C03638=1033.348,389.943,360.918,173.337,46.298,159.226
C03639=1033.357,390.188,360.876,173.346,46.301,159.228
C03640=1033.366,390.434,360.834,173.354,46.305,159.230
C03641=1033.376,390.680,360.790,173.364,46.308,159.232
C03642=1033.385,390.926,360.747,173.373,46.312,159.234
C03643=1033.394,391.173,360.704,173.381,46.316,159.236
C03644=1033.403,391.418,360.661,173.390,46.319,159.238
C03645=1033.413,391.665,360.617,173.399,46.323,159.240
C03646=1033.421,391.911,360.574,173.408,46.326,159.242
C03647=1033.431,392.156,360.531,173.417,46.330,159.244
C03648=1033.440,392.402,360.488,173.426,46.334,159.246
C03649=1033.450,392.649,360.445,173.435,46.337,159.248
C03650=1033.458,392.881,360.404,173.443,46.341,159.250
C03651=1033.467,393.113,360.362,173.452,46.345,159.252
C03652=1033.476,393.346,360.321,173.460,46.348,159.254
C03653=1033.485,393.578,360.281,173.469,46.352,159.256
C03654=1033.494,393.811,360.240,173.477,46.355,159.258
C03655=1033.502,394.044,360.198,173.486,46.359,159.260
C03656=1033.511,394.277,360.158,173.495,46.363,159.262
C03657=1033.521,394.509,360.116,173.505,46.366,159.264
C03658=1033.530,394.756,360.073,173.513,46.370,159.266
C03659=1033.539,395.001,360.029,173.522,46.374,159.268
C03660=1033.548,395.247,359.985,173.532,46.377,159.270
C03661=1033.558,395.493,359.941,173.541,46.381,159.272
C03662=1033.568,395.739,359.897,173.551,46.385,159.274
C03663=1033.577,395.984,359.854,173.560,46.389,159.276
C03664=1033.587,396.230,359.810,173.569,46.393,159.278
C03665=1033.596,396.476,359.766,173.578,46.397,159.280
C03666=1033.606,396.723,359.722,173.587,46.401,159.282
C03667=1033.614,396.968,359.678,173.597,46.405,159.285
C03668=1033.625,397.214,359.635,173.606,46.409,159.287
C03669=1033.634,397.460,359.590,173.616,46.413,159.289
C03670=1033.644,397.705,359.546,173.626,46.416,159.291
C03671=1033.654,397.951,359.502,173.635,46.421,159.293
C03672=1033.663,398.197,359.458,173.645,46.424,159.296
C03673=1033.673,398.443,359.413,173.654,46.429,159.298
C03674=1033.682,398.689,359.369,173.664,46.433,159.300
C03675=1033.692,398.935,359.326,173.673,46.437,159.302
C03676=1033.702,399.180,359.281,173.683,46.441,159.304
C03677=1033.712,399.427,359.237,173.693,46.445,159.307
C03678=1033.721,399.672,359.192,173.702,46.449,159.309
C03679=1033.731,399.918,359.148,173.712,46.453,159.311
C03680=1033.740,400.164,359.103,173.722,46.457,159.313
C03681=1033.751,400.410,359.059,173.731,46.462,159.316
C03682=1033.760,400.655,359.015,173.742,46.466,159.318
C03683=1033.770,400.901,358.970,173.752,46.470,159.320
C03684=1033.780,401.146,358.925,173.761,46.475,159.323
C03685=1033.790,401.393,358.880,173.771,46.479,159.325
C03686=1033.799,401.638,358.836,173.781,46.483,159.327
C03687=1033.809,401.884,358.791,173.791,46.487,159.330
C03688=1033.819,402.129,358.746,173.802,46.491,159.332
C03689=1033.829,402.375,358.701,173.811,46.496,159.334
C03690=1033.839,402.621,358.656,173.821,46.500,159.337
C03691=1033.849,402.867,358.611,173.831,46.505,159.339
C03692=1033.858,403.112,358.566,173.841,46.508,159.341
C03693=1033.867,403.358,358.521,173.852,46.513,159.344
C03694=1033.878,403.604,358.475,173.861,46.518,159.346
C03695=1033.888,403.849,358.430,173.871,46.522,159.348
C03696=1033.897,404.095,358.385,173.882,46.527,159.351
C03697=1033.908,404.341,358.340,173.892,46.531,159.353
C03698=1033.918,404.586,358.295,173.902,46.535,159.356
C03699=1033.928,404.832,358.249,173.913,46.540,159.358
C03700=1033.937,405.078,358.204,173.923,46.544,159.361
C03701=1033.947,405.323,358.158,173.933,46.549,159.363
C03702=1033.957,405.569,358.113,173.944,46.553,159.365
C03703=1033.967,405.814,358.068,173.954,46.558,159.368
C03704=1033.978,406.060,358.023,173.965,46.563,159.371
C03705=1033.988,406.306,357.976,173.975,46.567,159.373
C03706=1033.997,406.551,357.931,173.985,46.572,159.375
C03707=1034.008,406.797,357.885,173.996,46.576,159.378
C03708=1034.018,407.042,357.840,174.006,46.581,159.380
C03709=1034.029,407.287,357.794,174.017,46.585,159.383
C03710=1034.039,407.531,357.749,174.027,46.590,159.386
C03711=1034.049,407.773,357.704,174.038,46.595,159.388
C03712=1034.059,408.017,357.658,174.048,46.599,159.390
C03713=1034.069,408.259,357.613,174.059,46.604,159.393
C03714=1034.079,408.503,357.568,174.069,46.609,159.396
C03715=1034.089,408.745,357.523,174.080,46.614,159.398
C03716=1034.100,408.988,357.477,174.091,46.618,159.401
C03717=1034.110,409.231,357.431,174.102,46.623,159.403
C03718=1034.121,409.476,357.385,174.112,46.628,159.406
C03719=1034.130,409.722,357.339,174.123,46.633,159.409
C03720=1034.141,409.967,357.293,174.134,46.638,159.411
C03721=1034.151,410.213,357.247,174.145,46.642,159.414
C03722=1034.162,410.458,357.201,174.156,46.647,159.416
C03723=1034.172,410.704,357.154,174.166,46.652,159.419
C03724=1034.183,410.949,357.108,174.178,46.656,159.422
C03725=1034.193,411.195,357.062,174.189,46.662,159.424
C03726=1034.204,411.440,357.015,174.200,46.667,159.427
C03727=1034.214,411.686,356.969,174.211,46.671,159.430
C03728=1034.224,411.931,356.922,174.222,46.676,159.432
C03729=1034.235,412.176,356.876,174.234,46.681,159.435
C03730=1034.245,412.422,356.829,174.245,46.686,159.438
C03731=1034.257,412.668,356.782,174.255,46.691,159.441
C03732=1034.267,412.913,356.735,174.267,46.697,159.444
C03733=1034.277,413.159,356.689,174.278,46.701,159.446
C03734=1034.288,413.404,356.642,174.290,46.707,159.449
C03735=1034.298,413.649,356.594,174.301,46.712,159.452
C03736=1034.309,413.894,356.548,174.313,46.717,159.455
C03737=1034.320,414.140,356.500,174.325,46.722,159.458
C03738=1034.331,414.385,356.454,174.336,46.727,159.460
C03739=1034.341,414.630,356.406,174.347,46.732,159.463
C03740=1034.352,414.875,356.360,174.358,46.738,159.466
C03741=1034.362,415.121,356.312,174.370,46.743,159.469
C03742=1034.373,415.366,356.266,174.382,46.748,159.472
C03743=1034.384,415.612,356.218,174.393,46.753,159.475
C03744=1034.395,415.857,356.171,174.405,46.758,159.477
C03745=1034.406,416.102,356.123,174.417,46.764,159.480
C03746=1034.417,416.348,356.076,174.429,46.769,159.483
C03747=1034.427,416.593,356.029,174.441,46.774,159.486
C03748=1034.438,416.838,355.981,174.453,46.780,159.489
C03749=1034.449,417.083,355.934,174.465,46.785,159.492
C03750=1034.460,417.329,355.887,174.477,46.790,159.495
C03751=1034.471,417.574,355.839,174.488,46.796,159.498
C03752=1034.482,417.819,355.791,174.500,46.801,159.501
C03753=1034.493,418.064,355.744,174.513,46.807,159.504
C03754=1034.504,418.309,355.696,174.525,46.812,159.507
C03755=1034.514,418.554,355.648,174.537,46.818,159.510
C03756=1034.525,418.800,355.599,174.549,46.823,159.513
C03757=1034.537,419.045,355.552,174.561,46.829,159.516
C03758=1034.547,419.290,355.504,174.574,46.834,159.519
C03759=1034.558,419.535,355.456,174.586,46.840,159.522
C03760=1034.570,419.781,355.408,174.598,46.846,159.525
C03761=1034.581,420.026,355.360,174.610,46.851,159.528
C03762=1034.591,420.271,355.312,174.623,46.856,159.531
C03763=1034.603,420.515,355.263,174.635,46.862,159.535
C03764=1034.614,420.760,355.215,174.647,46.868,159.538
C03765=1034.625,421.006,355.167,174.660,46.874,159.541
C03766=1034.637,421.251,355.118,174.672,46.880,159.544
C03767=1034.648,421.497,355.070,174.685,46.885,159.547
C03768=1034.660,421.741,355.022,174.697,46.891,159.550
C03769=1034.670,421.986,354.974,174.711,46.897,159.554
C03770=1034.682,422.236,354.924,174.723,46.902,159.557
C03771=1034.693,422.485,354.874,174.736,46.909,159.560
C03772=1034.706,422.735,354.825,174.750,46.915,159.564
C03773=1034.717,422.985,354.775,174.762,46.920,159.567
C03774=1034.728,423.230,354.726,174.776,46.926,159.570
C03775=1034.739,423.475,354.678,174.788,46.932,159.573
C03776=1034.751,423.720,354.629,174.801,46.938,159.576
C03777=1034.762,423.965,354.580,174.814,46.944,159.580
C03778=1034.774,424.210,354.531,174.827,46.950,159.583
C03779=1034.786,424.455,354.482,174.840,46.956,159.587
C03780=1034.797,424.700,354.433,174.854,46.962,159.590
C03781=1034.809,424.944,354.384,174.866,46.968,159.593
C03782=1034.820,425.189,354.335,174.880,46.974,159.597
C03783=1034.832,425.434,354.285,174.893,46.980,159.600
C03784=1034.843,425.679,354.236,174.906,46.986,159.603
C03785=1034.854,425.924,354.187,174.919,46.992,159.607
C03786=1034.866,426.169,354.137,174.933,46.998,159.610
C03787=1034.878,426.414,354.088,174.947,47.004,159.614
C03788=1034.889,426.659,354.039,174.960,47.011,159.617
C03789=1034.901,426.903,353.988,174.974,47.016,159.621
C03790=1034.913,427.148,353.939,174.988,47.023,159.624
C03791=1034.925,427.394,353.890,175.000,47.029,159.627
C03792=1034.937,427.638,353.840,175.014,47.035,159.631
C03793=1034.948,427.883,353.790,175.028,47.042,159.635
C03794=1034.960,428.128,353.740,175.042,47.047,159.638
C03795=1034.972,428.372,353.691,175.055,47.054,159.642
C03796=1034.984,428.617,353.640,175.069,47.060,159.645
C03797=1034.995,428.862,353.590,175.083,47.067,159.649
C03798=1035.007,429.106,353.540,175.097,47.073,159.652
C03799=1035.019,429.351,353.490,175.111,47.079,159.656
C03800=1035.031,429.596,353.440,175.126,47.086,159.660
C03801=1035.043,429.841,353.390,175.140,47.092,159.663
C03802=1035.055,430.085,353.339,175.154,47.099,159.667
C03803=1035.066,430.330,353.289,175.168,47.105,159.671
C03804=1035.079,430.574,353.238,175.182,47.112,159.674
C03805=1035.091,430.819,353.188,175.196,47.118,159.678
C03806=1035.104,431.064,353.138,175.211,47.125,159.682
C03807=1035.115,431.308,353.087,175.225,47.132,159.686
C03808=1035.128,431.553,353.037,175.239,47.138,159.689
C03809=1035.140,431.796,352.986,175.254,47.145,159.693
C03810=1035.151,432.042,352.935,175.268,47.152,159.697
C03811=1035.164,432.286,352.885,175.284,47.158,159.701
C03812=1035.176,432.531,352.835,175.298,47.164,159.704
C03813=1035.188,432.775,352.783,175.312,47.171,159.708
C03814=1035.201,433.020,352.732,175.327,47.178,159.712
C03815=1035.214,433.265,352.682,175.342,47.185,159.716
C03816=1035.226,433.509,352.631,175.357,47.192,159.720
C03817=1035.238,433.754,352.580,175.372,47.198,159.724
C03818=1035.251,433.998,352.529,175.386,47.205,159.727
C03819=1035.264,434.243,352.478,175.402,47.212,159.732
C03820=1035.276,434.487,352.426,175.417,47.219,159.735
C03821=1035.289,434.731,352.375,175.432,47.226,159.739
C03822=1035.301,434.975,352.323,175.447,47.232,159.743
C03823=1035.314,435.220,352.272,175.463,47.239,159.747
C03824=1035.326,435.465,352.221,175.477,47.247,159.751
C03825=1035.339,435.708,352.169,175.493,47.253,159.755
C03826=1035.351,435.954,352.117,175.508,47.260,159.759
C03827=1035.364,436.197,352.066,175.523,47.267,159.763
C03828=1035.376,436.442,352.015,175.539,47.274,159.767
C03829=1035.390,436.686,351.963,175.555,47.281,159.772
C03830=1035.402,436.935,351.909,175.571,47.289,159.776
C03831=1035.415,437.183,351.857,175.587,47.296,159.780
C03832=1035.428,437.432,351.805,175.603,47.303,159.784
C03833=1035.441,437.680,351.751,175.619,47.310,159.788
C03834=1035.454,437.924,351.700,175.634,47.318,159.793
C03835=1035.466,438.169,351.647,175.650,47.325,159.797
C03836=1035.479,438.413,351.595,175.666,47.332,159.801
C03837=1035.492,438.657,351.543,175.682,47.339,159.805
C03838=1035.505,438.901,351.490,175.698,47.347,159.810
C03839=1035.519,439.145,351.438,175.714,47.354,159.814
C03840=1035.532,439.390,351.386,175.731,47.361,159.818
C03841=1035.544,439.633,351.333,175.747,47.369,159.822
C03842=1035.558,439.877,351.281,175.764,47.376,159.827
C03843=1035.570,440.122,351.228,175.780,47.384,159.831
C03844=1035.583,440.366,351.175,175.796,47.391,159.835
C03845=1035.597,440.609,351.123,175.812,47.398,159.840
C03846=1035.610,440.854,351.070,175.829,47.406,159.844
C03847=1035.623,441.098,351.017,175.846,47.413,159.849
C03848=1035.636,441.342,350.964,175.862,47.421,159.853
C03849=1035.650,441.585,350.911,175.879,47.428,159.857
C03850=1035.663,441.829,350.858,175.896,47.436,159.862
C03851=1035.676,442.073,350.805,175.913,47.444,159.867
C03852=1035.689,442.317,350.751,175.930,47.451,159.871
C03853=1035.703,442.561,350.699,175.947,47.458,159.875
C03854=1035.717,442.806,350.645,175.963,47.466,159.880
C03855=1035.730,443.050,350.592,175.981,47.474,159.885
C03856=1035.743,443.293,350.538,175.999,47.482,159.889
C03857=1035.757,443.537,350.486,176.015,47.490,159.894
C03858=1035.771,443.780,350.432,176.033,47.497,159.899
C03859=1035.785,444.023,350.378,176.050,47.505,159.903
C03860=1035.799,444.267,350.326,176.067,47.513,159.908
C03861=1035.813,444.510,350.274,176.085,47.520,159.912
C03862=1035.828,444.753,350.221,176.102,47.528,159.917
C03863=1035.844,444.996,350.169,176.121,47.535,159.922
C03864=1035.861,445.240,350.118,176.138,47.542,159.926
C03865=1035.877,445.484,350.067,176.156,47.550,159.931
C03866=1035.894,445.727,350.017,176.174,47.557,159.935
C03867=1035.913,445.971,349.967,176.191,47.564,159.940
C03868=1035.931,446.215,349.918,176.210,47.571,159.944
C03869=1035.949,446.460,349.869,176.228,47.577,159.949
C03870=1035.969,446.704,349.820,176.247,47.584,159.954
C03871=1035.989,446.948,349.772,176.265,47.591,159.958
C03872=1036.009,447.193,349.724,176.283,47.598,159.963
C03873=1036.031,447.437,349.677,176.301,47.604,159.967
C03874=1036.052,447.681,349.630,176.320,47.611,159.971
C03875=1036.075,447.926,349.583,176.339,47.617,159.976
C03876=1036.097,448.170,349.538,176.357,47.623,159.980
C03877=1036.120,448.415,349.492,176.376,47.629,159.985
C03878=1036.144,448.660,349.447,176.395,47.636,159.989
C03879=1036.168,448.905,349.402,176.414,47.642,159.994
C03880=1036.192,449.150,349.359,176.434,47.648,159.998
C03881=1036.218,449.395,349.314,176.452,47.653,160.002
C03882=1036.244,449.640,349.271,176.471,47.659,160.007
C03883=1036.271,449.885,349.228,176.492,47.665,160.011
C03884=1036.297,450.130,349.185,176.510,47.670,160.016
C03885=1036.325,450.376,349.144,176.531,47.676,160.020
C03886=1036.352,450.621,349.102,176.549,47.682,160.024
C03887=1036.382,450.866,349.061,176.569,47.687,160.029
C03888=1036.410,451.112,349.020,176.589,47.692,160.033
C03889=1036.440,451.357,348.980,176.609,47.698,160.037
C03890=1036.473,451.633,348.935,176.631,47.703,160.042
C03891=1036.509,451.908,348.891,176.654,47.709,160.047
C03892=1036.544,452.183,348.848,176.677,47.715,160.052
C03893=1036.579,452.458,348.805,176.699,47.720,160.057
C03894=1036.290,452.515,348.480,176.702,47.790,160.079
C03895=1036.256,452.253,348.521,176.681,47.785,160.074
C03896=1036.222,451.991,348.562,176.659,47.780,160.070
C03897=1036.188,451.729,348.604,176.638,47.775,160.065
C03898=1036.157,451.467,348.646,176.616,47.769,160.060
C03899=1036.127,451.222,348.686,176.596,47.764,160.056
C03900=1036.097,450.976,348.726,176.576,47.759,160.052
C03901=1036.068,450.730,348.768,176.557,47.754,160.047
C03902=1036.040,450.484,348.809,176.537,47.748,160.043
C03903=1036.012,450.240,348.850,176.517,47.743,160.039
C03904=1035.985,449.995,348.893,176.498,47.737,160.034
C03905=1035.958,449.750,348.936,176.478,47.732,160.030
C03906=1035.932,449.504,348.979,176.459,47.726,160.026
C03907=1035.907,449.259,349.022,176.440,47.720,160.021
C03908=1035.881,449.014,349.066,176.421,47.715,160.017
C03909=1035.857,448.769,349.111,176.402,47.709,160.012
C03910=1035.833,448.524,349.156,176.383,47.703,160.008
C03911=1035.810,448.279,349.201,176.363,47.697,160.003
C03912=1035.786,448.034,349.246,176.344,47.690,159.999
C03913=1035.764,447.790,349.292,176.326,47.684,159.994
C03914=1035.742,447.546,349.339,176.307,47.678,159.990
C03915=1035.721,447.302,349.386,176.289,47.671,159.986
C03916=1035.700,447.057,349.433,176.270,47.665,159.981
C03917=1035.680,446.812,349.481,176.251,47.659,159.977
C03918=1035.660,446.569,349.530,176.233,47.652,159.972
C03919=1035.641,446.324,349.578,176.215,47.645,159.968
C03920=1035.622,446.080,349.628,176.197,47.638,159.963
C03921=1035.604,445.836,349.678,176.179,47.631,159.958
C03922=1035.587,445.593,349.728,176.160,47.624,159.954
C03923=1035.569,445.349,349.778,176.143,47.618,159.949
C03924=1035.553,445.104,349.829,176.125,47.610,159.945
C03925=1035.537,444.861,349.881,176.107,47.603,159.940
C03926=1035.521,444.618,349.933,176.089,47.596,159.936
C03927=1035.506,444.374,349.985,176.072,47.588,159.931
C03928=1035.491,444.131,350.037,176.054,47.581,159.926
C03929=1035.477,443.888,350.090,176.037,47.573,159.922
C03930=1035.464,443.646,350.143,176.020,47.565,159.917
C03931=1035.450,443.402,350.197,176.002,47.557,159.912
C03932=1035.436,443.158,350.251,175.985,47.550,159.908
C03933=1035.423,442.914,350.304,175.967,47.542,159.903
C03934=1035.410,442.670,350.357,175.951,47.535,159.899
C03935=1035.396,442.426,350.410,175.933,47.528,159.894
C03936=1035.383,442.181,350.464,175.917,47.520,159.890
C03937=1035.369,441.938,350.517,175.899,47.512,159.885
C03938=1035.356,441.694,350.569,175.883,47.504,159.881
C03939=1035.343,441.450,350.623,175.866,47.497,159.876
C03940=1035.330,441.206,350.676,175.849,47.490,159.872
C03941=1035.316,440.962,350.728,175.832,47.483,159.867
C03942=1035.303,440.718,350.782,175.816,47.475,159.863
C03943=1035.290,440.474,350.834,175.800,47.468,159.859
C03944=1035.277,440.230,350.887,175.782,47.460,159.854
C03945=1035.263,439.986,350.940,175.766,47.453,159.850
C03946=1035.251,439.742,350.992,175.750,47.446,159.845
C03947=1035.238,439.498,351.045,175.733,47.438,159.841
C03948=1035.224,439.254,351.097,175.718,47.431,159.837
C03949=1035.211,439.009,351.150,175.700,47.424,159.833
C03950=1035.199,438.765,351.202,175.684,47.417,159.828
C03951=1035.185,438.520,351.254,175.668,47.409,159.824
C03952=1035.173,438.277,351.307,175.652,47.403,159.820
C03953=1035.159,438.033,351.359,175.636,47.395,159.815
C03954=1035.146,437.788,351.411,175.620,47.388,159.811
C03955=1035.134,437.539,351.464,175.604,47.381,159.807
C03956=1035.120,437.290,351.517,175.588,47.374,159.803
C03957=1035.107,437.040,351.570,175.572,47.366,159.799
C03958=1035.095,436.790,351.623,175.556,47.360,159.795
C03959=1035.081,436.546,351.675,175.541,47.353,159.790
C03960=1035.069,436.302,351.727,175.525,47.346,159.786
C03961=1035.056,436.057,351.778,175.510,47.339,159.782
C03962=1035.044,435.813,351.830,175.494,47.332,159.778
C03963=1035.031,435.569,351.881,175.478,47.325,159.774
C03964=1035.018,435.324,351.933,175.463,47.318,159.770
C03965=1035.006,435.080,351.984,175.448,47.311,159.766
C03966=1034.994,434.836,352.036,175.432,47.304,159.762
C03967=1034.980,434.591,352.087,175.418,47.297,159.758
C03968=1034.968,434.347,352.139,175.402,47.290,159.754
C03969=1034.956,434.103,352.190,175.388,47.284,159.750
C03970=1034.943,433.857,352.241,175.372,47.277,159.746
C03971=1034.931,433.612,352.292,175.358,47.270,159.743
C03972=1034.918,433.368,352.342,175.342,47.264,159.739
C03973=1034.906,433.124,352.393,175.328,47.257,159.735
C03974=1034.894,432.880,352.445,175.312,47.251,159.731
C03975=1034.881,432.635,352.496,175.298,47.244,159.727
C03976=1034.869,432.391,352.546,175.284,47.237,159.723
C03977=1034.857,432.146,352.597,175.268,47.231,159.719
C03978=1034.844,431.902,352.648,175.254,47.224,159.716
C03979=1034.832,431.657,352.698,175.240,47.218,159.712
C03980=1034.820,431.413,352.749,175.225,47.211,159.708
C03981=1034.808,431.168,352.799,175.211,47.205,159.705
C03982=1034.795,430.923,352.850,175.196,47.198,159.701
C03983=1034.783,430.679,352.900,175.181,47.192,159.697
C03984=1034.771,430.434,352.951,175.167,47.185,159.693
C03985=1034.760,430.189,353.001,175.153,47.179,159.690
C03986=1034.747,429.945,353.051,175.139,47.172,159.686
C03987=1034.736,429.699,353.102,175.125,47.166,159.682
C03988=1034.724,429.456,353.152,175.111,47.160,159.679
C03989=1034.711,429.211,353.202,175.096,47.153,159.675
C03990=1034.699,428.966,353.251,175.082,47.147,159.671
C03991=1034.688,428.721,353.302,175.068,47.141,159.668
C03992=1034.676,428.476,353.352,175.054,47.135,159.664
C03993=1034.664,428.232,353.402,175.041,47.128,159.661
C03994=1034.653,427.987,353.452,175.027,47.122,159.657
C03995=1034.640,427.742,353.502,175.013,47.115,159.654
C03996=1034.629,427.498,353.551,174.999,47.110,159.650
C03997=1034.617,427.253,353.601,174.985,47.103,159.647
C03998=1034.605,427.008,353.651,174.973,47.097,159.643
C03999=1034.593,426.763,353.701,174.958,47.091,159.640
C04000=1034.582,426.518,353.750,174.945,47.085,159.636
C04001=1034.570,426.273,353.800,174.932,47.079,159.633
C04002=1034.559,426.029,353.849,174.918,47.073,159.629
C04003=1034.547,425.784,353.898,174.904,47.067,159.626
C04004=1034.535,425.538,353.948,174.891,47.061,159.622
C04005=1034.524,425.294,353.997,174.878,47.055,159.619
C04006=1034.512,425.049,354.046,174.865,47.049,159.616
C04007=1034.501,424.804,354.095,174.851,47.043,159.612
C04008=1034.489,424.559,354.144,174.838,47.037,159.609
C04009=1034.478,424.314,354.193,174.825,47.031,159.606
C04010=1034.466,424.069,354.242,174.812,47.025,159.602
C04011=1034.455,423.825,354.291,174.799,47.020,159.599
C04012=1034.443,423.580,354.340,174.786,47.013,159.596
C04013=1034.432,423.335,354.389,174.774,47.008,159.593
C04014=1034.421,423.090,354.437,174.760,47.002,159.589
C04015=1034.409,422.838,354.488,174.747,46.996,159.586
C04016=1034.397,422.586,354.538,174.733,46.990,159.583
C04017=1034.385,422.333,354.588,174.720,46.985,159.579
C04018=1034.373,422.082,354.637,174.707,46.978,159.576
C04019=1034.362,421.837,354.686,174.695,46.973,159.573
C04020=1034.351,421.592,354.735,174.681,46.967,159.569
C04021=1034.340,421.346,354.783,174.669,46.961,159.566
C04022=1034.328,421.102,354.832,174.656,46.956,159.563
C04023=1034.317,420.857,354.880,174.644,46.950,159.560
C04024=1034.306,420.611,354.928,174.632,46.944,159.557
C04025=1034.294,420.366,354.976,174.619,46.939,159.554
C04026=1034.283,420.120,355.024,174.607,46.933,159.551
C04027=1034.273,419.876,355.072,174.594,46.928,159.548
C04028=1034.262,419.630,355.121,174.581,46.923,159.545
C04029=1034.250,419.385,355.168,174.569,46.917,159.541
C04030=1034.239,419.140,355.217,174.557,46.911,159.538
C04031=1034.228,418.895,355.265,174.545,46.906,159.535
C04032=1034.217,418.650,355.313,174.532,46.901,159.532
C04033=1034.207,418.405,355.361,174.520,46.895,159.529
C04034=1034.195,418.160,355.409,174.509,46.889,159.526
C04035=1034.184,417.914,355.456,174.497,46.884,159.523
C04036=1034.174,417.670,355.504,174.484,46.879,159.520
C04037=1034.162,417.424,355.552,174.472,46.874,159.517
C04038=1034.152,417.179,355.600,174.460,46.868,159.514
C04039=1034.140,416.934,355.647,174.448,46.863,159.511
C04040=1034.130,416.689,355.694,174.436,46.858,159.508
C04041=1034.119,416.443,355.741,174.425,46.852,159.506
C04042=1034.108,416.197,355.789,174.413,46.847,159.503
C04043=1034.097,415.953,355.836,174.401,46.842,159.500
C04044=1034.087,415.707,355.884,174.389,46.837,159.497
C04045=1034.075,415.462,355.931,174.377,46.832,159.494
C04046=1034.065,415.216,355.978,174.366,46.826,159.491
C04047=1034.054,414.970,356.025,174.354,46.822,159.488
C04048=1034.043,414.725,356.072,174.342,46.816,159.485
C04049=1034.033,414.481,356.120,174.331,46.811,159.483
C04050=1034.022,414.235,356.166,174.319,46.806,159.480
C04051=1034.011,413.989,356.213,174.308,46.801,159.477
C04052=1034.000,413.744,356.260,174.296,46.796,159.474
C04053=1033.990,413.499,356.307,174.285,46.791,159.471
C04054=1033.979,413.254,356.354,174.273,46.786,159.468
C04055=1033.969,413.009,356.401,174.262,46.781,159.466
C04056=1033.957,412.763,356.448,174.251,46.775,159.463
C04057=1033.947,412.517,356.495,174.239,46.771,159.460
C04058=1033.937,412.272,356.541,174.228,46.766,159.458
C04059=1033.926,412.027,356.588,174.216,46.761,159.455
C04060=1033.916,411.781,356.634,174.206,46.756,159.452
C04061=1033.906,411.536,356.682,174.195,46.751,159.449
C04062=1033.895,411.290,356.727,174.183,46.746,159.447
C04063=1033.885,411.045,356.775,174.173,46.741,159.444
C04064=1033.874,410.799,356.821,174.161,46.737,159.441
C04065=1033.863,410.554,356.866,174.150,46.732,159.439
C04066=1033.854,410.308,356.913,174.139,46.727,159.436
C04067=1033.843,410.063,356.960,174.128,46.722,159.433
C04068=1033.832,409.817,357.005,174.117,46.717,159.431
C04069=1033.821,409.572,357.051,174.106,46.712,159.428
C04070=1033.811,409.326,357.097,174.095,46.708,159.425
C04071=1033.801,409.083,357.143,174.084,46.703,159.423
C04072=1033.791,408.838,357.189,174.074,46.699,159.420
C04073=1033.781,408.595,357.234,174.063,46.694,159.418
C04074=1033.770,408.350,357.280,174.053,46.689,159.415
C04075=1033.760,408.107,357.326,174.041,46.685,159.413
C04076=1033.750,407.863,357.371,174.031,46.680,159.410
C04077=1033.739,407.619,357.416,174.020,46.675,159.407
C04078=1033.730,407.375,357.462,174.010,46.671,159.405
C04079=1033.719,407.129,357.507,173.999,46.667,159.403
C04080=1033.709,406.884,357.553,173.989,46.662,159.400
C04081=1033.699,406.639,357.599,173.978,46.657,159.397
C04082=1033.688,406.392,357.644,173.968,46.653,159.395
C04083=1033.679,406.147,357.690,173.957,46.649,159.393
C04084=1033.669,405.901,357.735,173.946,46.644,159.390
C04085=1033.659,405.656,357.781,173.936,46.639,159.387
C04086=1033.648,405.410,357.826,173.925,46.635,159.385
C04087=1033.638,405.165,357.872,173.915,46.630,159.383
C04088=1033.628,404.919,357.917,173.905,46.626,159.380
C04089=1033.619,404.674,357.963,173.894,46.621,159.378
C04090=1033.608,404.427,358.008,173.884,46.617,159.375
C04091=1033.599,404.182,358.053,173.875,46.613,159.373
C04092=1033.588,403.936,358.099,173.864,46.608,159.371
C04093=1033.578,403.691,358.144,173.854,46.604,159.368
C04094=1033.569,403.445,358.189,173.844,46.599,159.366
C04095=1033.560,403.199,358.234,173.833,46.595,159.363
C04096=1033.549,402.953,358.279,173.823,46.591,159.361
C04097=1033.540,402.708,358.324,173.813,46.587,159.359
C04098=1033.530,402.462,358.369,173.803,46.582,159.356
C04099=1033.520,402.216,358.414,173.794,46.578,159.354
C04100=1033.510,401.970,358.459,173.783,46.574,159.351
C04101=1033.500,401.725,358.504,173.773,46.570,159.349
C04102=1033.490,401.479,358.549,173.763,46.566,159.347
C04103=1033.481,401.234,358.593,173.753,46.561,159.345
C04104=1033.471,400.988,358.638,173.744,46.557,159.342
C04105=1033.461,400.742,358.683,173.734,46.553,159.340
C04106=1033.451,400.496,358.727,173.723,46.549,159.338
C04107=1033.441,400.251,358.772,173.713,46.545,159.335
C04108=1033.431,400.005,358.816,173.704,46.541,159.333
C04109=1033.422,399.759,358.861,173.694,46.537,159.331
C04110=1033.412,399.514,358.905,173.684,46.532,159.329
C04111=1033.403,399.268,358.950,173.675,46.528,159.326
C04112=1033.393,399.022,358.994,173.665,46.524,159.324
C04113=1033.383,398.776,359.038,173.655,46.520,159.322
C04114=1033.373,398.530,359.082,173.646,46.516,159.320
C04115=1033.364,398.285,359.127,173.636,46.513,159.318
C04116=1033.354,398.038,359.171,173.626,46.509,159.315
C04117=1033.344,397.793,359.214,173.617,46.505,159.313
C04118=1033.335,397.547,359.259,173.607,46.501,159.311
C04119=1033.325,397.301,359.303,173.598,46.496,159.309
C04120=1033.315,397.056,359.347,173.588,46.493,159.307
C04121=1033.306,396.810,359.391,173.578,46.489,159.305
C04122=1033.297,396.564,359.435,173.569,46.485,159.302
C04123=1033.286,396.318,359.478,173.559,46.481,159.300
C04124=1033.277,396.072,359.522,173.551,46.477,159.298
C04125=1033.268,395.826,359.566,173.541,46.473,159.296
C04126=1033.259,395.580,359.610,173.532,46.470,159.294
C04127=1033.249,395.334,359.654,173.522,46.466,159.292
C04128=1033.239,395.088,359.698,173.513,46.462,159.290
C04129=1033.230,394.843,359.742,173.504,46.458,159.287
C04130=1033.220,394.597,359.785,173.495,46.455,159.285
C04131=1033.212,394.363,359.826,173.486,46.451,159.283
C04132=1033.203,394.129,359.868,173.477,46.447,159.281
C04133=1033.194,393.895,359.910,173.468,46.444,159.279
C04134=1033.184,393.661,359.950,173.460,46.441,159.278
C04135=1033.176,393.428,359.992,173.451,46.437,159.276
C04136=1033.167,393.195,360.033,173.443,46.433,159.274
C04137=1033.158,392.960,360.074,173.434,46.430,159.272
C04138=1033.149,392.727,360.115,173.425,46.426,159.270
C04139=1033.140,392.481,360.159,173.416,46.423,159.268
C04140=1033.130,392.235,360.202,173.407,46.419,159.266
C04141=1033.121,391.989,360.245,173.398,46.416,159.264
C04142=1033.112,391.743,360.288,173.389,46.412,159.262
C04143=1033.103,391.497,360.332,173.380,46.409,159.260
C04144=1033.093,391.251,360.374,173.371,46.405,159.258
C04145=1033.084,391.005,360.417,173.362,46.402,159.256
C04146=1033.074,390.759,360.461,173.353,46.398,159.254
C04147=1033.066,390.513,360.504,173.344,46.394,159.252
C04148=1033.057,390.267,360.546,173.335,46.391,159.250
C04149=1033.047,390.020,360.590,173.327,46.387,159.248
C04150=1033.038,389.775,360.632,173.317,46.384,159.246
C04151=1033.028,389.528,360.675,173.309,46.380,159.244
C04152=1033.020,389.282,360.718,173.300,46.377,159.242
C04153=1033.011,389.036,360.760,173.292,46.374,159.240
C04154=1033.001,388.790,360.803,173.283,46.370,159.239
C04155=1032.992,388.544,360.846,173.274,46.367,159.236
C04156=1032.983,388.298,360.889,173.265,46.363,159.235
C04157=1032.975,388.052,360.932,173.256,46.360,159.233
C04158=1032.965,387.806,360.975,173.248,46.357,159.231
C04159=1032.956,387.560,361.017,173.239,46.353,159.229
C04160=1032.947,387.313,361.059,173.231,46.350,159.227
C04161=1032.938,387.067,361.102,173.222,46.347,159.225
C04162=1032.928,386.821,361.145,173.214,46.343,159.223
C04163=1032.919,386.575,361.186,173.206,46.340,159.222
C04164=1032.910,386.329,361.229,173.196,46.337,159.220
C04165=1032.901,386.082,361.270,173.187,46.334,159.218
C04166=1032.892,385.837,361.313,173.179,46.331,159.216
C04167=1032.883,385.590,361.355,173.171,46.327,159.214
C04168=1032.873,385.344,361.397,173.162,46.324,159.212
C04169=1032.865,385.097,361.440,173.154,46.321,159.211
C04170=1032.856,384.851,361.481,173.146,46.318,159.209
C04171=1032.847,384.605,361.524,173.137,46.315,159.207
C04172=1032.838,384.359,361.566,173.129,46.312,159.205
C04173=1032.829,384.112,361.607,173.120,46.309,159.203
C04174=1032.820,383.867,361.650,173.112,46.305,159.202
C04175=1032.811,383.620,361.691,173.104,46.302,159.200
C04176=1032.802,383.374,361.733,173.095,46.299,159.198
C04177=1032.793,383.128,361.775,173.087,46.296,159.196
C04178=1032.784,382.881,361.817,173.080,46.293,159.195
C04179=1032.775,382.635,361.858,173.071,46.290,159.193
C04180=1032.766,382.389,361.901,173.063,46.287,159.191
C04181=1032.757,382.143,361.942,173.055,46.284,159.189
C04182=1032.748,381.896,361.984,173.047,46.281,159.188
C04183=1032.740,381.650,362.026,173.038,46.278,159.186
C04184=1032.731,381.404,362.068,173.030,46.275,159.184
C04185=1032.722,381.158,362.109,173.022,46.272,159.183
C04186=1032.714,380.911,362.150,173.014,46.269,159.181
C04187=1032.705,380.664,362.192,173.006,46.266,159.179
C04188=1032.696,380.418,362.234,172.998,46.263,159.178
C04189=1032.688,380.172,362.275,172.990,46.260,159.176
C04190=1032.679,379.926,362.317,172.982,46.257,159.174
C04191=1032.671,379.709,362.353,172.974,46.255,159.173
C04192=1032.664,379.493,362.390,172.968,46.252,159.171
C04193=1032.656,379.277,362.426,172.961,46.249,159.170
C04194=1032.648,379.061,362.463,172.954,46.247,159.168
C04195=1032.640,378.845,362.498,172.947,46.244,159.167
C04196=1032.634,378.629,362.535,172.940,46.242,159.165
C04197=1032.626,378.413,362.572,172.933,46.239,159.164
C04198=1032.618,378.196,362.607,172.926,46.237,159.163
C04199=1032.610,377.950,362.649,172.918,46.234,159.161
C04200=1032.601,377.704,362.690,172.911,46.231,159.159
C04201=1032.592,377.457,362.731,172.903,46.228,159.158
C04202=1032.584,377.211,362.772,172.895,46.226,159.156
C04203=1032.575,376.964,362.812,172.888,46.223,159.154
C04204=1032.566,376.718,362.854,172.879,46.220,159.153
C04205=1032.558,376.472,362.895,172.871,46.218,159.151
C04206=1032.548,376.225,362.935,172.863,46.215,159.150
C04207=1032.540,375.979,362.976,172.856,46.212,159.148
C04208=1032.531,375.732,363.018,172.848,46.210,159.147
C04209=1032.523,375.486,363.058,172.841,46.207,159.145
C04210=1032.514,375.239,363.099,172.833,46.204,159.143
C04211=1032.505,374.992,363.140,172.825,46.202,159.142
C04212=1032.497,374.746,363.180,172.818,46.199,159.140
C04213=1032.488,374.499,363.221,172.810,46.197,159.139
C04214=1032.480,374.253,363.261,172.802,46.194,159.137
C04215=1032.472,374.007,363.302,172.795,46.191,159.136
C04216=1032.463,373.760,363.342,172.787,46.189,159.134
C04217=1032.455,373.514,363.383,172.780,46.186,159.133
C04218=1032.446,373.267,363.424,172.772,46.184,159.131
C04219=1032.438,373.021,363.465,172.765,46.181,159.130
C04220=1032.429,372.775,363.505,172.757,46.178,159.128
C04221=1032.420,372.528,363.546,172.750,46.176,159.127
C04222=1032.413,372.281,363.586,172.742,46.173,159.125
C04223=1032.403,372.034,363.626,172.735,46.170,159.124
C04224=1032.395,371.788,363.667,172.727,46.168,159.122
C04225=1032.387,371.541,363.707,172.720,46.165,159.121
C04226=1032.379,371.295,363.747,172.713,46.163,159.119
C04227=1032.370,371.048,363.788,172.705,46.161,159.118
C04228=1032.362,370.802,363.828,172.698,46.158,159.116
C04229=1032.354,370.555,363.868,172.691,46.156,159.115
C04230=1032.346,370.309,363.908,172.683,46.154,159.113
C04231=1032.337,370.062,363.949,172.676,46.151,159.112
C04232=1032.329,369.815,363.989,172.668,46.149,159.110
C04233=1032.321,369.569,364.029,172.661,46.146,159.109
C04234=1032.313,369.322,364.069,172.654,46.143,159.108
C04235=1032.304,369.075,364.108,172.646,46.141,159.106
C04236=1032.295,368.829,364.149,172.640,46.139,159.105
C04237=1032.287,368.582,364.189,172.632,46.136,159.103
C04238=1032.279,368.335,364.228,172.625,46.134,159.102
C04239=1032.267,367.992,364.284,172.615,46.131,159.100
C04240=1032.256,367.647,364.339,172.605,46.128,159.098
C04241=1032.244,367.303,364.394,172.595,46.125,159.096
C04242=1032.232,366.959,364.450,172.585,46.121,159.094
C04243=1032.224,366.712,364.490,172.578,46.119,159.093
C04244=1032.216,366.466,364.530,172.570,46.117,159.091
C04245=1032.207,366.219,364.569,172.564,46.115,159.090
C04246=1032.200,365.972,364.609,172.557,46.112,159.089
C04247=1032.191,365.725,364.648,172.549,46.110,159.087
C04248=1032.183,365.479,364.687,172.542,46.108,159.086
C04249=1032.175,365.232,364.727,172.536,46.106,159.085
C04250=1032.167,364.985,364.767,172.528,46.104,159.083
C04251=1032.156,364.672,364.817,172.520,46.101,159.082
C04252=1032.146,364.357,364.867,172.511,46.099,159.080
C04253=1032.136,364.044,364.917,172.501,46.096,159.078
C04254=1032.125,363.730,364.967,172.493,46.093,159.077
C04255=1032.117,363.483,365.007,172.486,46.091,159.075
C04256=1032.109,363.236,365.046,172.479,46.089,159.074
C04257=1032.101,362.989,365.085,172.472,46.087,159.073
C04258=1032.093,362.742,365.125,172.466,46.084,159.071
C04259=1032.085,362.495,365.164,172.458,46.082,159.070
C04260=1032.077,362.249,365.202,172.451,46.081,159.069
C04261=1032.069,362.002,365.242,172.445,46.078,159.067
C04262=1032.061,361.755,365.281,172.438,46.076,159.066
C04263=1032.053,361.508,365.320,172.431,46.074,159.065
C04264=1032.044,361.262,365.359,172.425,46.072,159.064
C04265=1032.037,361.015,365.398,172.417,46.070,159.062
C04266=1032.029,360.768,365.438,172.410,46.068,159.061
C04267=1032.021,360.521,365.476,172.404,46.066,159.060
C04268=1032.012,360.274,365.515,172.397,46.064,159.059
C04269=1032.005,360.028,365.554,172.391,46.062,159.057
C04270=1031.997,359.781,365.592,172.384,46.061,159.056
C04271=1031.988,359.534,365.632,172.377,46.059,159.055
C04272=1031.980,359.287,365.670,172.370,46.057,159.054
C04273=1031.973,359.040,365.708,172.364,46.055,159.052
C04274=1031.964,358.793,365.747,172.357,46.053,159.051
C04275=1031.956,358.547,365.786,172.350,46.051,159.050
C04276=1031.948,358.300,365.825,172.344,46.049,159.049
C04277=1031.940,358.053,365.863,172.338,46.047,159.048
C04278=1031.932,357.806,365.902,172.331,46.045,159.046
C04279=1031.925,357.559,365.940,172.324,46.043,159.045
C04280=1031.916,357.312,365.979,172.318,46.042,159.044
C04281=1031.908,357.065,366.017,172.310,46.040,159.043
C04282=1031.901,356.818,366.056,172.304,46.038,159.042
C04283=1031.893,356.571,366.094,172.297,46.037,159.040
C04284=1031.885,356.324,366.132,172.291,46.035,159.039
C04285=1031.877,356.077,366.171,172.285,46.033,159.038
C04286=1031.869,355.831,366.209,172.278,46.031,159.037
C04287=1031.861,355.583,366.248,172.271,46.029,159.036
C04288=1031.854,355.337,366.286,172.265,46.027,159.034
C04289=1031.845,355.090,366.325,172.258,46.025,159.033
C04290=1031.837,354.842,366.363,172.252,46.024,159.032
C04291=1031.830,354.596,366.402,172.246,46.023,159.031
C04292=1031.821,354.348,366.439,172.239,46.021,159.030
C04293=1031.814,354.102,366.477,172.233,46.019,159.029
C04294=1031.805,353.855,366.516,172.226,46.017,159.028
C04295=1031.798,353.608,366.553,172.220,46.016,159.027
C04296=1031.791,353.361,366.592,172.214,46.014,159.025
C04297=1031.782,353.114,366.630,172.207,46.013,159.024
C04298=1031.775,352.867,366.667,172.201,46.011,159.023
C04299=1031.766,352.620,366.706,172.194,46.009,159.022
C04300=1031.759,352.373,366.743,172.188,46.007,159.021
C04301=1031.750,352.126,366.781,172.182,46.006,159.020
C04302=1031.743,351.879,366.819,172.175,46.004,159.019
C04303=1031.735,351.632,366.857,172.170,46.002,159.018
C04304=1031.727,351.385,366.896,172.163,46.001,159.017
C04305=1031.720,351.138,366.933,172.157,45.999,159.016
C04306=1031.712,350.891,366.970,172.151,45.998,159.014
C04307=1031.700,350.485,367.032,172.141,45.995,159.013
C04308=1031.687,350.081,367.094,172.130,45.993,159.011
C04309=1031.675,349.675,367.156,172.120,45.990,159.009
C04310=1031.661,349.270,367.218,172.110,45.988,159.007
C04311=1031.654,349.023,367.256,172.104,45.986,159.006
C04312=1031.646,348.777,367.293,172.097,45.985,159.005
C04313=1031.639,348.530,367.331,172.091,45.983,159.004
C04314=1031.631,348.282,367.369,172.085,45.982,159.003
C04315=1031.623,348.035,367.406,172.079,45.980,159.002
C04316=1031.616,347.788,367.443,172.074,45.979,159.001
C04317=1031.608,347.541,367.480,172.067,45.977,159.000
C04318=1031.600,347.294,367.518,172.061,45.976,158.999
C04319=1031.592,347.046,367.555,172.055,45.975,158.998
C04320=1031.585,346.799,367.593,172.049,45.974,158.997
C04321=1031.577,346.552,367.629,172.042,45.972,158.996
C04322=1031.569,346.305,367.667,172.037,45.971,158.995
C04323=1031.561,346.058,367.704,172.031,45.969,158.994
C04324=1031.554,345.811,367.741,172.025,45.968,158.993
C04325=1031.546,345.564,367.778,172.018,45.966,158.992
C04326=1031.539,345.317,367.816,172.013,45.965,158.991
C04327=1031.530,345.070,367.853,172.007,45.964,158.990
C04328=1031.523,344.822,367.890,172.001,45.963,158.989
C04329=1031.515,344.575,367.927,171.995,45.961,158.988
C04330=1031.508,344.328,367.964,171.988,45.960,158.987
C04331=1031.500,344.081,368.001,171.983,45.958,158.986
C04332=1031.493,343.834,368.039,171.977,45.957,158.985
C04333=1031.485,343.587,368.075,171.971,45.956,158.984
C04334=1031.478,343.339,368.113,171.964,45.955,158.983
C04335=1031.470,343.093,368.150,171.959,45.953,158.982
C04336=1031.462,342.845,368.186,171.953,45.952,158.981
C04337=1031.455,342.598,368.223,171.947,45.951,158.980
C04338=1031.447,342.351,368.260,171.942,45.949,158.979
C04339=1031.440,342.103,368.297,171.936,45.948,158.978
C04340=1031.432,341.857,368.334,171.929,45.947,158.977
C04341=1031.425,341.610,368.370,171.924,45.946,158.976
C04342=1031.418,341.363,368.407,171.918,45.945,158.976
C04343=1031.410,341.115,368.444,171.912,45.944,158.975
C04344=1031.403,340.868,368.481,171.906,45.943,158.974
C04345=1031.395,340.621,368.517,171.901,45.941,158.973
C04346=1031.388,340.373,368.554,171.895,45.940,158.972
C04347=1031.380,340.126,368.591,171.889,45.939,158.971
C04348=1031.372,339.879,368.627,171.884,45.938,158.970
C04349=1031.365,339.631,368.664,171.878,45.937,158.969
C04350=1031.358,339.385,368.700,171.871,45.936,158.968
C04351=1031.350,339.138,368.736,171.866,45.935,158.967
C04352=1031.342,338.890,368.773,171.860,45.934,158.966
C04353=1031.335,338.643,368.809,171.854,45.932,158.965
C04354=1031.327,338.395,368.845,171.849,45.932,158.965
C04355=1031.320,338.148,368.883,171.843,45.930,158.964
C04356=1031.313,337.902,368.918,171.837,45.929,158.963
C04357=1031.305,337.654,368.955,171.832,45.928,158.962
C04358=1031.297,337.407,368.991,171.826,45.927,158.961
C04359=1031.290,337.159,369.027,171.821,45.926,158.960
C04360=1031.283,336.912,369.063,171.815,45.925,158.959
C04361=1031.276,336.665,369.100,171.809,45.924,158.958
C04362=1031.268,336.417,369.136,171.804,45.923,158.957
C04363=1031.255,336.009,369.196,171.794,45.921,158.956
C04364=1031.243,335.601,369.256,171.785,45.919,158.954
C04365=1031.231,335.193,369.315,171.776,45.918,158.953
C04366=1031.220,334.784,369.375,171.767,45.916,158.952
C04367=1031.212,334.537,369.411,171.761,45.915,158.951
C04368=1031.204,334.289,369.447,171.756,45.914,158.950
C04369=1031.197,334.042,369.483,171.750,45.914,158.949
C04370=1031.190,333.794,369.519,171.744,45.913,158.948
C04371=1031.183,333.548,369.554,171.739,45.912,158.948
C04372=1031.175,333.300,369.591,171.733,45.911,158.947
C04373=1031.167,333.053,369.626,171.728,45.910,158.946
C04374=1031.160,332.806,369.661,171.722,45.909,158.945
C04375=1031.152,332.558,369.698,171.717,45.908,158.944
C04376=1031.145,332.311,369.733,171.712,45.908,158.943
C04377=1031.138,332.063,369.769,171.707,45.907,158.943
C04378=1031.130,331.816,369.805,171.700,45.906,158.942
C04379=1031.123,331.569,369.840,171.696,45.905,158.941
C04380=1031.116,331.321,369.877,171.690,45.904,158.940
C04381=1031.108,331.074,369.912,171.685,45.903,158.939
C04382=1031.100,330.827,369.947,171.679,45.903,158.939
C04383=1031.093,330.580,369.983,171.674,45.902,158.938
C04384=1031.086,330.332,370.019,171.668,45.901,158.937
C04385=1031.079,330.085,370.055,171.663,45.900,158.936
C04386=1031.071,329.837,370.090,171.657,45.899,158.935
C04387=1031.065,329.590,370.125,171.652,45.898,158.935
C04388=1031.057,329.342,370.161,171.646,45.898,158.934
C04389=1031.050,329.095,370.196,171.642,45.897,158.933
C04390=1031.042,328.848,370.232,171.636,45.896,158.932
C04391=1031.035,328.600,370.267,171.631,45.895,158.932
C04392=1031.028,328.353,370.302,171.625,45.895,158.931
C04393=1031.021,328.106,370.339,171.620,45.894,158.930
C04394=1031.014,327.858,370.374,171.615,45.893,158.929
C04395=1031.006,327.611,370.408,171.609,45.892,158.928
C04396=1030.999,327.363,370.444,171.604,45.892,158.928
C04397=1030.991,327.116,370.478,171.599,45.892,158.927
C04398=1030.984,326.868,370.514,171.594,45.891,158.926
C04399=1030.976,326.622,370.549,171.588,45.890,158.926
C04400=1030.970,326.374,370.584,171.583,45.889,158.925
C04401=1030.961,326.126,370.619,171.578,45.889,158.924
C04402=1030.955,325.879,370.654,171.573,45.888,158.923
C04403=1030.947,325.631,370.689,171.567,45.888,158.923
C04404=1030.939,325.384,370.724,171.562,45.887,158.922
C04405=1030.932,325.137,370.759,171.557,45.887,158.921
C04406=1030.924,324.889,370.794,171.552,45.886,158.921
C04407=1030.917,324.642,370.829,171.547,45.885,158.920
C04408=1030.910,324.394,370.863,171.541,45.885,158.919
C04409=1030.903,324.146,370.898,171.536,45.884,158.918
C04410=1030.895,323.899,370.933,171.531,45.884,158.918
C04411=1030.888,323.652,370.967,171.526,45.884,158.917
C04412=1030.881,323.405,371.002,171.521,45.883,158.916
C04413=1030.873,323.157,371.037,171.515,45.882,158.915
C04414=1030.866,322.909,371.072,171.510,45.882,158.915
C04415=1030.859,322.662,371.106,171.505,45.881,158.914
C04416=1030.852,322.414,371.141,171.500,45.881,158.914
C04417=1030.845,322.167,371.176,171.495,45.880,158.913
C04418=1030.837,321.920,371.211,171.489,45.880,158.912
C04419=1030.825,321.507,371.269,171.481,45.879,158.911
C04420=1030.813,321.094,371.326,171.473,45.878,158.910
C04421=1030.801,320.681,371.385,171.465,45.877,158.909
C04422=1030.789,320.267,371.442,171.456,45.877,158.908
C04423=1030.782,320.020,371.476,171.451,45.876,158.907
C04424=1030.775,319.773,371.511,171.446,45.876,158.906
C04425=1030.768,319.525,371.545,171.441,45.875,158.906
C04426=1030.761,319.278,371.580,171.435,45.875,158.905
C04427=1030.754,319.030,371.614,171.431,45.875,158.904
C04428=1030.746,318.783,371.649,171.426,45.874,158.904
C04429=1030.740,318.535,371.683,171.420,45.874,158.903
C04430=1030.732,318.288,371.718,171.416,45.873,158.902
C04431=1030.726,318.040,371.752,171.411,45.873,158.902
C04432=1030.718,317.793,371.787,171.406,45.872,158.901
C04433=1030.711,317.545,371.820,171.401,45.872,158.901
C04434=1030.704,317.298,371.856,171.396,45.871,158.900
C04435=1030.697,317.050,371.889,171.391,45.871,158.899
C04436=1030.690,316.803,371.924,171.387,45.871,158.899
C04437=1030.683,316.555,371.958,171.381,45.870,158.898
C04438=1030.676,316.308,371.992,171.376,45.870,158.897
C04439=1030.669,316.060,372.027,171.372,45.870,158.897
C04440=1030.662,315.813,372.061,171.367,45.869,158.896
C04441=1030.655,315.565,372.095,171.361,45.869,158.895
C04442=1030.648,315.318,372.130,171.357,45.869,158.895
C04443=1030.641,315.070,372.164,171.352,45.868,158.894
C04444=1030.634,314.822,372.198,171.347,45.868,158.893
C04445=1030.627,314.576,372.233,171.342,45.868,158.893
C04446=1030.620,314.328,372.266,171.337,45.867,158.892
C04447=1030.614,314.080,372.301,171.332,45.867,158.892
C04448=1030.607,313.832,372.335,171.328,45.867,158.891
C04449=1030.599,313.585,372.368,171.323,45.867,158.891
C04450=1030.593,313.337,372.404,171.317,45.866,158.890
C04451=1030.586,313.090,372.437,171.313,45.866,158.889
C04452=1030.579,312.843,372.471,171.308,45.865,158.889
C04453=1030.572,312.595,372.505,171.304,45.865,158.888
C04454=1030.565,312.347,372.539,171.299,45.865,158.887
C04455=1030.558,312.099,372.573,171.294,45.865,158.887
C04456=1030.552,311.852,372.607,171.289,45.865,158.886
C04457=1030.545,311.605,372.642,171.284,45.864,158.886
C04458=1030.537,311.357,372.675,171.279,45.864,158.885
C04459=1030.532,311.110,372.709,171.275,45.863,158.884
C04460=1030.524,310.862,372.742,171.270,45.864,158.884
C04461=1030.517,310.614,372.776,171.266,45.863,158.883
C04462=1030.510,310.367,372.810,171.260,45.863,158.883
C04463=1030.502,310.119,372.843,171.256,45.863,158.882
C04464=1030.494,309.872,372.877,171.251,45.863,158.882
C04465=1030.488,309.624,372.909,171.247,45.863,158.881
C04466=1030.481,309.376,372.943,171.241,45.863,158.881
C04467=1030.474,309.129,372.977,171.236,45.863,158.880
C04468=1030.466,308.881,373.010,171.232,45.863,158.879
C04469=1030.459,308.634,373.043,171.228,45.863,158.879
C04470=1030.452,308.386,373.077,171.223,45.863,158.879
C04471=1030.445,308.138,373.110,171.218,45.863,158.878
C04472=1030.437,307.890,373.143,171.213,45.863,158.877
C04473=1030.431,307.643,373.177,171.208,45.863,158.877
C04474=1030.424,307.395,373.210,171.204,45.863,158.876
C04475=1030.413,306.987,373.265,171.196,45.862,158.875
C04476=1030.400,306.580,373.319,171.188,45.862,158.875
C04477=1030.389,306.171,373.374,171.181,45.863,158.874
C04478=1030.377,305.763,373.429,171.174,45.862,158.873
C04479=1030.371,305.516,373.462,171.169,45.862,158.872
C04480=1030.363,305.268,373.495,171.164,45.863,158.872
C04481=1030.356,305.021,373.528,171.159,45.862,158.871
C04482=1030.349,304.773,373.561,171.155,45.863,158.871
C04483=1030.343,304.524,373.594,171.150,45.863,158.870
C04484=1030.335,304.278,373.627,171.146,45.862,158.870
C04485=1030.328,304.030,373.660,171.141,45.863,158.869
C04486=1030.322,303.783,373.694,171.137,45.862,158.869
C04487=1030.315,303.534,373.727,171.132,45.863,158.868
C04488=1030.308,303.287,373.759,171.128,45.863,158.868
C04489=1030.301,303.039,373.793,171.123,45.863,158.867
C04490=1030.294,302.792,373.826,171.118,45.863,158.867
C04491=1030.287,302.544,373.858,171.114,45.863,158.866
C04492=1030.280,302.295,373.891,171.109,45.863,158.866
C04493=1030.273,302.048,373.925,171.105,45.863,158.865
C04494=1030.267,301.801,373.957,171.100,45.863,158.865
C04495=1030.259,301.553,373.990,171.096,45.863,158.865
C04496=1030.253,301.305,374.023,171.091,45.863,158.864
C04497=1030.246,301.058,374.057,171.087,45.863,158.864
C04498=1030.239,300.810,374.089,171.082,45.863,158.863
C04499=1030.232,300.562,374.122,171.078,45.864,158.863
C04500=1030.225,300.314,374.155,171.074,45.864,158.862
C04501=1030.218,300.066,374.187,171.069,45.864,158.862
C04502=1030.211,299.819,374.221,171.065,45.864,158.861
C04503=1030.204,299.571,374.254,171.060,45.864,158.861
C04504=1030.198,299.324,374.286,171.056,45.864,158.860
C04505=1030.191,299.076,374.319,171.051,45.864,158.860
C04506=1030.184,298.828,374.352,171.047,45.864,158.859
C04507=1030.178,298.580,374.384,171.043,45.865,158.859
C04508=1030.171,298.333,374.417,171.038,45.864,158.858
C04509=1030.164,298.085,374.450,171.034,45.865,158.858
C04510=1030.158,297.837,374.482,171.029,45.865,158.857
C04511=1030.151,297.590,374.515,171.025,45.865,158.857
C04512=1030.144,297.342,374.548,171.020,45.865,158.857
C04513=1030.137,297.094,374.580,171.016,45.865,158.856
C04514=1030.130,296.847,374.613,171.012,45.866,158.856
C04515=1030.123,296.599,374.646,171.007,45.866,158.855
C04516=1030.117,296.351,374.678,171.003,45.866,158.855
C04517=1030.110,296.104,374.711,170.999,45.866,158.854
C04518=1030.103,295.855,374.744,170.994,45.866,158.854
C04519=1030.097,295.608,374.776,170.990,45.866,158.853
C04520=1030.091,295.360,374.808,170.985,45.867,158.853
C04521=1030.084,295.112,374.841,170.981,45.867,158.853
C04522=1030.077,294.864,374.874,170.976,45.867,158.852
C04523=1030.071,294.616,374.906,170.972,45.867,158.852
C04524=1030.064,294.369,374.939,170.968,45.867,158.851
C04525=1030.057,294.122,374.971,170.963,45.868,158.851
C04526=1030.050,293.873,375.003,170.959,45.868,158.850
C04527=1030.043,293.626,375.035,170.955,45.869,158.850
C04528=1030.037,293.377,375.067,170.951,45.869,158.850
C04529=1030.030,293.130,375.099,170.946,45.869,158.849
C04530=1030.022,292.882,375.132,170.943,45.869,158.849
C04531=1030.012,292.491,375.183,170.935,45.870,158.848
C04532=1030.001,292.100,375.233,170.929,45.870,158.847
C04533=1029.991,291.709,375.283,170.922,45.871,158.847
C04534=1029.979,291.318,375.334,170.916,45.871,158.846
C04535=1029.973,291.070,375.366,170.912,45.872,158.846
C04536=1029.966,290.822,375.398,170.907,45.872,158.846
C04537=1029.959,290.575,375.430,170.903,45.873,158.845
C04538=1029.953,290.327,375.461,170.899,45.873,158.845
C04539=1029.946,290.080,375.493,170.894,45.874,158.844
C04540=1029.939,289.831,375.526,170.890,45.874,158.844
C04541=1029.932,289.583,375.557,170.886,45.874,158.844
C04542=1029.925,289.336,375.589,170.881,45.875,158.843
C04543=1029.919,289.088,375.621,170.877,45.875,158.843
C04544=1029.912,288.840,375.654,170.873,45.875,158.842
C04545=1029.906,288.593,375.685,170.869,45.876,158.842
C04546=1029.899,288.345,375.717,170.864,45.877,158.842
C04547=1029.891,288.096,375.748,170.860,45.877,158.841
C04548=1029.884,287.849,375.780,170.857,45.877,158.841
C04549=1029.878,287.601,375.812,170.853,45.877,158.841
C04550=1029.871,287.353,375.843,170.848,45.878,158.840
C04551=1029.864,287.105,375.875,170.844,45.879,158.840
C04552=1029.858,286.857,375.907,170.840,45.879,158.840
C04553=1029.851,286.610,375.939,170.836,45.879,158.839
C04554=1029.845,286.362,375.970,170.831,45.880,158.839
C04555=1029.838,286.114,376.002,170.827,45.881,158.839
C04556=1029.831,285.866,376.033,170.823,45.881,158.838
C04557=1029.824,285.618,376.065,170.820,45.881,158.838
C04558=1029.818,285.370,376.096,170.815,45.882,158.838
C04559=1029.810,285.121,376.128,170.811,45.883,158.837
C04560=1029.804,284.874,376.159,170.807,45.883,158.837
C04561=1029.797,284.626,376.191,170.803,45.884,158.837
C04562=1029.789,284.378,376.222,170.798,45.884,158.836
C04563=1029.783,284.130,376.253,170.794,45.885,158.836
C04564=1029.776,283.882,376.284,170.790,45.886,158.836
C04565=1029.769,283.634,376.316,170.786,45.886,158.835
C04566=1029.762,283.386,376.347,170.783,45.887,158.835
C04567=1029.756,283.139,376.379,170.778,45.887,158.835
C04568=1029.749,282.891,376.410,170.774,45.888,158.834
C04569=1029.742,282.643,376.442,170.770,45.888,158.834
C04570=1029.736,282.395,376.473,170.766,45.889,158.834
C04571=1029.729,282.147,376.504,170.762,45.890,158.833
C04572=1029.721,281.899,376.535,170.757,45.890,158.833
C04573=1029.715,281.651,376.567,170.754,45.891,158.833
C04574=1029.708,281.403,376.597,170.750,45.891,158.832
C04575=1029.702,281.155,376.629,170.746,45.892,158.832
C04576=1029.695,280.908,376.660,170.742,45.892,158.832
C04577=1029.689,280.660,376.691,170.738,45.893,158.831
C04578=1029.682,280.412,376.723,170.733,45.894,158.831
C04579=1029.676,280.163,376.754,170.730,45.895,158.831
C04580=1029.669,279.916,376.785,170.726,45.895,158.830
C04581=1029.662,279.668,376.816,170.722,45.896,158.830
C04582=1029.655,279.420,376.847,170.718,45.896,158.830
C04583=1029.648,279.172,376.878,170.714,45.897,158.830
C04584=1029.641,278.924,376.909,170.710,45.898,158.829
C04585=1029.635,278.676,376.941,170.706,45.898,158.829
C04586=1029.629,278.428,376.971,170.702,45.899,158.829
C04587=1029.618,278.050,377.019,170.696,45.900,158.828
C04588=1029.609,277.670,377.066,170.690,45.901,158.828
C04589=1029.598,277.291,377.114,170.683,45.902,158.827
C04590=1029.588,276.913,377.161,170.678,45.903,158.827
C04591=1029.581,276.665,377.191,170.674,45.904,158.827
C04592=1029.574,276.417,377.223,170.670,45.905,158.826
C04593=1029.568,276.169,377.253,170.666,45.905,158.826
C04594=1029.561,275.921,377.283,170.662,45.906,158.826
C04595=1029.554,275.673,377.315,170.659,45.907,158.826
C04596=1029.547,275.424,377.345,170.655,45.908,158.825
C04597=1029.541,275.177,377.376,170.650,45.908,158.825
C04598=1029.534,274.929,377.407,170.646,45.909,158.825
C04599=1029.527,274.681,377.438,170.642,45.910,158.825
C04600=1029.520,274.433,377.468,170.639,45.911,158.824
C04601=1029.515,274.185,377.499,170.635,45.911,158.824
C04602=1029.507,273.937,377.529,170.631,45.912,158.824
C04603=1029.501,273.689,377.560,170.627,45.913,158.824
C04604=1029.494,273.440,377.590,170.624,45.914,158.823
C04605=1029.487,273.192,377.622,170.620,45.915,158.823
C04606=1029.481,272.945,377.652,170.615,45.915,158.823
C04607=1029.474,272.696,377.682,170.611,45.916,158.822
C04608=1029.467,272.449,377.714,170.607,45.917,158.822
C04609=1029.461,272.201,377.743,170.604,45.918,158.822
C04610=1029.454,271.953,377.774,170.600,45.919,158.822
C04611=1029.447,271.704,377.804,170.596,45.920,158.822
C04612=1029.440,271.456,377.836,170.592,45.921,158.821
C04613=1029.434,271.209,377.865,170.589,45.921,158.821
C04614=1029.427,270.960,377.896,170.585,45.922,158.821
C04615=1029.420,270.712,377.926,170.581,45.923,158.821
C04616=1029.414,270.464,377.957,170.577,45.924,158.820
C04617=1029.407,270.216,377.987,170.574,45.925,158.820
C04618=1029.400,269.968,378.018,170.570,45.926,158.820
C04619=1029.394,269.721,378.048,170.566,45.927,158.820
C04620=1029.387,269.472,378.079,170.562,45.928,158.819
C04621=1029.380,269.224,378.109,170.559,45.929,158.819
C04622=1029.374,268.976,378.139,170.554,45.930,158.819
C04623=1029.367,268.728,378.169,170.550,45.931,158.819
C04624=1029.360,268.480,378.199,170.547,45.931,158.819
C04625=1029.354,268.232,378.230,170.543,45.932,158.818
C04626=1029.347,267.984,378.260,170.539,45.933,158.818
C04627=1029.340,267.735,378.290,170.535,45.934,158.818
C04628=1029.334,267.488,378.320,170.532,45.935,158.818
C04629=1029.327,267.239,378.350,170.528,45.936,158.817
C04630=1029.321,266.992,378.380,170.524,45.937,158.817
C04631=1029.314,266.743,378.411,170.520,45.938,158.817
C04632=1029.307,266.495,378.440,170.517,45.939,158.817
C04633=1029.301,266.247,378.470,170.513,45.940,158.817
C04634=1029.294,265.999,378.501,170.509,45.941,158.816
C04635=1029.288,265.751,378.531,170.506,45.942,158.816
C04636=1029.281,265.503,378.561,170.502,45.943,158.816
C04637=1029.273,265.255,378.591,170.498,45.944,158.816
C04638=1029.267,265.006,378.620,170.494,45.945,158.816
C04639=1029.261,264.758,378.651,170.491,45.946,158.815
C04640=1029.254,264.510,378.680,170.487,45.947,158.815
C04641=1029.247,264.262,378.710,170.483,45.948,158.815
C04642=1029.240,264.015,378.740,170.480,45.949,158.815
C04643=1029.231,263.640,378.785,170.474,45.951,158.815
C04644=1029.220,263.266,378.830,170.468,45.952,158.814
C04645=1029.211,262.891,378.875,170.463,45.954,158.814
C04646=1029.200,262.518,378.920,170.457,45.955,158.814
C04647=1029.194,262.269,378.950,170.454,45.956,158.814
C04648=1029.188,262.022,378.980,170.450,45.957,158.813
C04649=1029.181,261.773,379.010,170.446,45.959,158.813
C04650=1029.174,261.525,379.039,170.443,45.959,158.813
C04651=1029.167,261.277,379.069,170.439,45.960,158.813
C04652=1029.162,261.029,379.100,170.435,45.961,158.813
C04653=1029.154,260.781,379.128,170.433,45.963,158.813
C04654=1029.148,260.533,379.157,170.429,45.964,158.812
C04655=1029.141,260.284,379.187,170.425,45.965,158.812
C04656=1029.134,260.036,379.217,170.421,45.966,158.812
C04657=1029.127,259.788,379.247,170.418,45.967,158.812
C04658=1029.120,259.540,379.275,170.414,45.969,158.812
C04659=1029.113,259.292,379.305,170.410,45.970,158.812
C04660=1029.107,259.044,379.334,170.407,45.971,158.812
C04661=1029.100,258.795,379.364,170.403,45.972,158.811
C04662=1029.093,258.548,379.393,170.399,45.974,158.811
C04663=1029.086,258.299,379.422,170.396,45.974,158.811
C04664=1029.079,258.051,379.451,170.392,45.976,158.811
C04665=1029.072,257.803,379.481,170.388,45.977,158.811
C04666=1029.066,257.555,379.510,170.385,45.979,158.811
C04667=1029.059,257.306,379.540,170.382,45.979,158.811
C04668=1029.052,257.058,379.569,170.378,45.981,158.811
C04669=1029.045,256.810,379.598,170.374,45.982,158.810
C04670=1029.039,256.562,379.627,170.371,45.983,158.810
C04671=1029.033,256.313,379.657,170.367,45.984,158.810
C04672=1029.025,256.065,379.687,170.363,45.986,158.810
C04673=1029.018,255.817,379.715,170.360,45.987,158.810
C04674=1029.012,255.569,379.744,170.356,45.988,158.810
C04675=1029.005,255.320,379.774,170.352,45.989,158.809
C04676=1028.999,255.072,379.803,170.350,45.991,158.809
C04677=1028.992,254.824,379.833,170.346,45.992,158.809
C04678=1028.985,254.576,379.861,170.342,45.993,158.809
C04679=1028.979,254.328,379.890,170.339,45.994,158.809
C04680=1028.972,254.079,379.920,170.335,45.996,158.809
C04681=1028.966,253.831,379.949,170.332,45.996,158.809
C04682=1028.959,253.583,379.978,170.328,45.998,158.809
C04683=1028.952,253.334,380.006,170.324,46.000,158.809
C04684=1028.945,253.087,380.036,170.321,46.000,158.808
C04685=1028.939,252.839,380.065,170.318,46.002,158.808
C04686=1028.932,252.590,380.095,170.314,46.003,158.808
C04687=1028.926,252.342,380.124,170.311,46.004,158.808
C04688=1028.919,252.094,380.152,170.307,46.006,158.808
C04689=1028.912,251.845,380.182,170.304,46.007,158.808
C04690=1028.906,251.597,380.211,170.300,46.008,158.808
C04691=1028.900,251.349,380.240,170.296,46.009,158.808
C04692=1028.893,251.101,380.268,170.294,46.011,158.808
C04693=1028.886,250.852,380.297,170.290,46.012,158.807
C04694=1028.879,250.604,380.327,170.287,46.013,158.807
C04695=1028.873,250.356,380.356,170.283,46.015,158.807
C04696=1028.866,250.108,380.384,170.279,46.016,158.807
C04697=1028.859,249.859,380.413,170.276,46.017,158.807
C04698=1028.853,249.611,380.442,170.272,46.019,158.807
C04699=1028.843,249.236,380.486,170.268,46.021,158.807
C04700=1028.834,248.860,380.530,170.262,46.023,158.807
C04701=1028.823,248.484,380.574,170.257,46.025,158.806
C04702=1028.813,248.109,380.618,170.252,46.026,158.806
C04703=1028.807,247.861,380.647,170.248,46.028,158.806
C04704=1028.801,247.612,380.675,170.244,46.029,158.806
C04705=1028.795,247.364,380.704,170.242,46.030,158.806
C04706=1028.787,247.116,380.733,170.238,46.032,158.806
C04707=1028.781,246.868,380.762,170.235,46.033,158.806
C04708=1028.775,246.619,380.791,170.231,46.034,158.806
C04709=1028.769,246.371,380.820,170.228,46.036,158.806
C04710=1028.762,246.123,380.848,170.225,46.037,158.806
C04711=1028.756,245.875,380.877,170.222,46.038,158.805
C04712=1028.749,245.627,380.906,170.218,46.040,158.805
C04713=1028.743,245.378,380.935,170.215,46.041,158.805
C04714=1028.736,245.130,380.964,170.211,46.042,158.805
C04715=1028.730,244.881,380.992,170.207,46.044,158.805
C04716=1028.723,244.633,381.021,170.204,46.045,158.805
C04717=1028.717,244.385,381.050,170.201,46.047,158.805
C04718=1028.710,244.137,381.078,170.198,46.048,158.805
C04719=1028.704,243.888,381.107,170.194,46.049,158.805
C04720=1028.697,243.641,381.135,170.191,46.051,158.805
C04721=1028.691,243.392,381.163,170.187,46.052,158.805
C04722=1028.684,243.143,381.192,170.185,46.054,158.805
C04723=1028.677,242.895,381.221,170.181,46.055,158.804
C04724=1028.671,242.647,381.249,170.178,46.057,158.804
C04725=1028.665,242.399,381.278,170.174,46.058,158.804
C04726=1028.658,242.150,381.306,170.171,46.060,158.804
C04727=1028.652,241.902,381.335,170.168,46.061,158.804
C04728=1028.645,241.654,381.363,170.164,46.062,158.804
C04729=1028.639,241.405,381.392,170.161,46.064,158.804
C04730=1028.632,241.157,381.419,170.157,46.065,158.804
C04731=1028.625,240.909,381.448,170.154,46.067,158.804
C04732=1028.619,240.660,381.476,170.151,46.068,158.804
C04733=1028.612,240.413,381.505,170.148,46.070,158.804
C04734=1028.606,240.164,381.533,170.144,46.071,158.804
C04735=1028.599,239.916,381.561,170.141,46.073,158.804
C04736=1028.592,239.668,381.589,170.138,46.074,158.804
C04737=1028.586,239.418,381.618,170.135,46.076,158.804
C04738=1028.579,239.170,381.646,170.131,46.077,158.804
C04739=1028.572,238.922,381.674,170.127,46.079,158.804
C04740=1028.566,238.673,381.702,170.125,46.080,158.804
C04741=1028.559,238.425,381.731,170.121,46.082,158.803
C04742=1028.553,238.177,381.758,170.118,46.083,158.803
C04743=1028.546,237.928,381.786,170.115,46.086,158.804
C04744=1028.539,237.681,381.815,170.112,46.087,158.803
C04745=1028.532,237.432,381.842,170.108,46.089,158.803
C04746=1028.526,237.183,381.871,170.105,46.090,158.803
C04747=1028.520,236.935,381.898,170.102,46.092,158.803
C04748=1028.513,236.687,381.927,170.099,46.093,158.803
C04749=1028.506,236.439,381.955,170.095,46.095,158.803
C04750=1028.499,236.190,381.982,170.091,46.096,158.803
C04751=1028.493,235.942,382.010,170.089,46.098,158.803
C04752=1028.487,235.693,382.038,170.085,46.100,158.803
C04753=1028.480,235.445,382.067,170.082,46.101,158.803
C04754=1028.473,235.197,382.095,170.078,46.103,158.803
C04755=1028.463,234.815,382.137,170.074,46.105,158.803
C04756=1028.453,234.434,382.180,170.068,46.108,158.803
C04757=1028.442,234.052,382.223,170.064,46.110,158.803
C04758=1028.433,233.671,382.266,170.059,46.113,158.803
C04759=1028.426,233.422,382.293,170.055,46.114,158.803
C04760=1028.420,233.174,382.321,170.053,46.116,158.803
C04761=1028.413,232.925,382.349,170.049,46.118,158.803
C04762=1028.406,232.677,382.376,170.046,46.119,158.803
C04763=1028.400,232.428,382.405,170.043,46.121,158.803
C04764=1028.394,232.180,382.433,170.040,46.122,158.803
C04765=1028.387,231.931,382.460,170.036,46.125,158.803
C04766=1028.381,231.683,382.488,170.034,46.126,158.803
C04767=1028.374,231.435,382.515,170.030,46.128,158.803
C04768=1028.367,231.187,382.543,170.027,46.129,158.803
C04769=1028.361,230.938,382.571,170.024,46.131,158.803
C04770=1028.354,230.690,382.599,170.021,46.133,158.803
C04771=1028.347,230.441,382.626,170.017,46.134,158.803
C04772=1028.341,230.193,382.654,170.014,46.136,158.803
C04773=1028.334,229.944,382.682,170.011,46.138,158.803
C04774=1028.328,229.697,382.709,170.008,46.139,158.803
C04775=1028.321,229.448,382.737,170.004,46.141,158.803
C04776=1028.315,229.200,382.765,170.002,46.143,158.803
C04777=1028.308,228.951,382.792,169.998,46.145,158.803
C04778=1028.301,228.703,382.820,169.995,46.146,158.803
C04779=1028.295,228.454,382.847,169.992,46.148,158.803
C04780=1028.289,228.206,382.874,169.989,46.150,158.803
C04781=1028.282,227.958,382.902,169.985,46.151,158.803
C04782=1028.275,227.709,382.930,169.983,46.153,158.803
C04783=1028.269,227.461,382.958,169.979,46.155,158.803
C04784=1028.262,227.212,382.985,169.977,46.157,158.803
C04785=1028.256,226.963,383.012,169.973,46.159,158.803
C04786=1028.249,226.716,383.039,169.970,46.160,158.803
C04787=1028.242,226.467,383.067,169.967,46.162,158.803
C04788=1028.236,226.218,383.094,169.964,46.164,158.803
C04789=1028.229,225.970,383.122,169.960,46.166,158.803
C04790=1028.222,225.722,383.149,169.958,46.167,158.803
C04791=1028.216,225.473,383.175,169.954,46.170,158.803
C04792=1028.209,225.225,383.203,169.951,46.171,158.803
C04793=1028.203,224.976,383.230,169.948,46.173,158.803
C04794=1028.195,224.728,383.257,169.945,46.175,158.803
C04795=1028.189,224.479,383.285,169.942,46.177,158.803
C04796=1028.183,224.231,383.312,169.939,46.178,158.803
C04797=1028.176,223.983,383.339,169.936,46.181,158.804
C04798=1028.169,223.734,383.366,169.933,46.182,158.803
C04799=1028.163,223.485,383.394,169.930,46.184,158.804
C04800=1028.156,223.238,383.421,169.926,46.186,158.804
C04801=1028.149,222.989,383.447,169.924,46.188,158.804
C04802=1028.143,222.740,383.475,169.920,46.190,158.804
C04803=1028.136,222.491,383.502,169.918,46.192,158.804
C04804=1028.130,222.244,383.529,169.914,46.194,158.804
C04805=1028.123,221.995,383.556,169.911,46.195,158.804
C04806=1028.116,221.746,383.584,169.908,46.198,158.804
C04807=1028.110,221.497,383.611,169.905,46.199,158.804
C04808=1028.104,221.250,383.638,169.902,46.201,158.804
C04809=1028.097,221.001,383.664,169.899,46.203,158.804
C04810=1028.090,220.752,383.692,169.896,46.205,158.804
C04811=1028.081,220.363,383.734,169.891,46.207,158.804
C04812=1028.070,219.974,383.776,169.887,46.211,158.804
C04813=1028.060,219.584,383.819,169.881,46.213,158.804
C04814=1028.049,219.195,383.862,169.877,46.217,158.804
C04815=1028.043,218.947,383.888,169.874,46.218,158.804
C04816=1028.036,218.698,383.915,169.871,46.220,158.805
C04817=1028.029,218.450,383.942,169.868,46.222,158.805
C04818=1028.023,218.202,383.968,169.865,46.224,158.805
C04819=1028.017,217.953,383.995,169.862,46.226,158.805
C04820=1028.009,217.705,384.023,169.859,46.228,158.805
C04821=1028.003,217.457,384.049,169.856,46.230,158.805
C04822=1027.996,217.208,384.076,169.852,46.232,158.805
C04823=1027.989,216.959,384.102,169.850,46.234,158.805
C04824=1027.983,216.711,384.129,169.846,46.236,158.805
C04825=1027.976,216.462,384.156,169.844,46.238,158.805
C04826=1027.970,216.213,384.183,169.840,46.240,158.805
C04827=1027.963,215.965,384.209,169.838,46.242,158.805
C04828=1027.957,215.716,384.236,169.835,46.244,158.805
C04829=1027.950,215.469,384.263,169.832,46.246,158.806
C04830=1027.943,215.220,384.289,169.829,46.248,158.806
C04831=1027.936,214.971,384.316,169.825,46.250,158.806
C04832=1027.930,214.723,384.342,169.823,46.252,158.806
C04833=1027.923,214.474,384.369,169.819,46.254,158.806
C04834=1027.917,214.226,384.395,169.817,46.256,158.806
C04835=1027.910,213.977,384.423,169.813,46.258,158.806
C04836=1027.903,213.729,384.449,169.811,46.260,158.806
C04837=1027.897,213.481,384.476,169.808,46.262,158.806
C04838=1027.890,213.231,384.503,169.805,46.264,158.806
C04839=1027.884,212.983,384.529,169.802,46.266,158.806
C04840=1027.877,212.734,384.556,169.799,46.268,158.806
C04841=1027.871,212.486,384.582,169.796,46.270,158.807
C04842=1027.864,212.237,384.609,169.794,46.272,158.807
C04843=1027.857,211.988,384.635,169.790,46.274,158.807
C04844=1027.851,211.741,384.662,169.787,46.276,158.807
C04845=1027.844,211.492,384.689,169.784,46.278,158.807
C04846=1027.838,211.244,384.715,169.781,46.280,158.807
C04847=1027.831,210.995,384.742,169.778,46.283,158.807
C04848=1027.825,210.747,384.768,169.775,46.285,158.807
C04849=1027.818,210.498,384.794,169.773,46.286,158.807
C04850=1027.812,210.250,384.821,169.769,46.288,158.807
C04851=1027.805,210.001,384.847,169.767,46.290,158.807
C04852=1027.798,209.753,384.874,169.763,46.293,158.807
C04853=1027.791,209.504,384.900,169.761,46.295,158.808
C04854=1027.786,209.255,384.926,169.758,46.297,158.808
C04855=1027.779,209.006,384.952,169.755,46.299,158.808
C04856=1027.772,208.758,384.978,169.752,46.301,158.808
C04857=1027.765,208.510,385.005,169.749,46.303,158.808
C04858=1027.759,208.261,385.031,169.746,46.306,158.808
C04859=1027.752,208.013,385.058,169.743,46.308,158.808
C04860=1027.746,207.764,385.084,169.740,46.310,158.808
C04861=1027.738,207.516,385.110,169.738,46.312,158.809
C04862=1027.732,207.267,385.136,169.734,46.314,158.809
C04863=1027.725,207.018,385.162,169.732,46.316,158.809
C04864=1027.719,206.770,385.189,169.729,46.319,158.809
C04865=1027.712,206.521,385.215,169.726,46.321,158.809
C04866=1027.706,206.273,385.241,169.723,46.323,158.809
C04867=1027.696,205.888,385.281,169.718,46.326,158.809
C04868=1027.685,205.504,385.321,169.714,46.329,158.810
C04869=1027.675,205.120,385.362,169.710,46.333,158.810
C04870=1027.664,204.734,385.402,169.705,46.336,158.810
C04871=1027.639,203.692,385.506,169.326,46.233,158.744
C04872=1027.634,203.443,385.530,169.323,46.236,158.745
C04873=1027.628,203.194,385.554,169.319,46.239,158.745
C04874=1027.622,202.945,385.580,169.314,46.242,158.745
C04875=1027.616,202.697,385.603,169.311,46.245,158.745
C04876=1027.609,202.449,385.629,169.307,46.248,158.745
C04877=1027.604,202.200,385.653,169.304,46.251,158.745
C04878=1027.598,201.951,385.678,169.299,46.253,158.745
C04879=1027.593,201.702,385.702,169.295,46.257,158.746
C04880=1027.587,201.453,385.727,169.292,46.260,158.746
C04881=1027.581,201.205,385.751,169.288,46.263,158.746
C04882=1027.575,200.956,385.776,169.284,46.266,158.746
C04883=1027.569,200.707,385.801,169.280,46.269,158.746
C04884=1027.563,200.459,385.825,169.277,46.271,158.747
C04885=1027.557,200.209,385.850,169.272,46.274,158.747
C04886=1027.551,199.961,385.873,169.268,46.278,158.747
C04887=1027.545,199.712,385.898,169.265,46.281,158.747
C04888=1027.539,199.463,385.922,169.261,46.284,158.747
C04889=1027.533,199.214,385.946,169.257,46.287,158.748
C04890=1027.527,198.966,385.970,169.253,46.290,158.748
C04891=1027.521,198.717,385.994,169.249,46.293,158.748
C04892=1027.516,198.468,386.018,169.246,46.296,158.748
C04893=1027.509,198.220,386.043,169.242,46.299,158.748
C04894=1027.503,197.971,386.067,169.239,46.303,158.749
C04895=1027.497,197.722,386.091,169.234,46.306,158.749
C04896=1027.491,197.474,386.116,169.230,46.309,158.749
C04897=1027.485,197.225,386.140,169.227,46.312,158.749
C04898=1027.480,196.976,386.163,169.223,46.316,158.749
C04899=1027.473,196.727,386.187,169.220,46.319,158.750
C04900=1027.467,196.478,386.211,169.215,46.322,158.750
C04901=1027.461,196.229,386.235,169.212,46.325,158.750
C04902=1027.455,195.981,386.259,169.208,46.328,158.750
C04903=1027.449,195.731,386.284,169.205,46.331,158.750
C04904=1027.443,195.483,386.307,169.200,46.334,158.751
C04905=1027.438,195.235,386.332,169.197,46.337,158.751
C04906=1027.431,194.986,386.356,169.193,46.340,158.751
C04907=1027.425,194.737,386.379,169.189,46.344,158.751
C04908=1027.419,194.488,386.404,169.185,46.346,158.751
C04909=1027.414,194.239,386.427,169.182,46.350,158.752
C04910=1027.408,193.991,386.451,169.178,46.353,158.752
C04911=1027.402,193.742,386.475,169.174,46.357,158.752
C04912=1027.396,193.493,386.499,169.171,46.360,158.752
C04913=1027.390,193.244,386.523,169.167,46.363,158.753
C04914=1027.384,192.996,386.547,169.163,46.366,158.753
C04915=1027.379,192.747,386.571,169.159,46.369,158.753
C04916=1027.372,192.498,386.595,169.156,46.372,158.753
C04917=1027.367,192.249,386.619,169.152,46.375,158.753
C04918=1027.361,192.001,386.643,169.149,46.378,158.754
C04919=1027.355,191.751,386.667,169.146,46.382,158.754
C04920=1027.349,191.503,386.690,169.141,46.385,158.754
C04921=1027.343,191.254,386.714,169.138,46.388,158.754
C04922=1027.337,191.005,386.738,169.134,46.391,158.755
C04923=1027.331,190.756,386.761,169.131,46.394,158.755
C04924=1027.326,190.507,386.786,169.126,46.397,158.755
C04925=1027.319,190.259,386.810,169.123,46.400,158.755
C04926=1027.314,190.010,386.833,169.119,46.404,158.755
C04927=1027.308,189.761,386.857,169.116,46.407,158.756
C04928=1027.302,189.513,386.881,169.112,46.410,158.756
C04929=1027.297,189.263,386.904,169.109,46.413,158.756
C04930=1027.291,189.015,386.928,169.105,46.416,158.756
C04931=1027.285,188.766,386.952,169.101,46.420,158.756
C04932=1027.279,188.483,386.979,169.097,46.423,158.757
C04933=1027.273,188.200,387.006,169.093,46.427,158.757
C04934=1027.265,187.917,387.033,169.089,46.431,158.757
C04935=1027.259,187.634,387.060,169.085,46.434,158.757
C04936=1027.253,187.385,387.083,169.082,46.437,158.758
C04937=1027.247,187.137,387.107,169.078,46.441,158.758
C04938=1027.242,186.888,387.131,169.075,46.444,158.758
C04939=1027.236,186.639,387.154,169.071,46.447,158.758
C04940=1027.230,186.390,387.179,169.067,46.450,158.759
C04941=1027.225,186.141,387.202,169.064,46.453,158.759
C04942=1027.219,185.893,387.225,169.061,46.456,158.759
C04943=1027.214,185.644,387.249,169.057,46.460,158.759
C04944=1027.208,185.395,387.272,169.053,46.463,158.760
C04945=1027.201,185.146,387.296,169.049,46.466,158.760
C04946=1027.196,184.897,387.320,169.046,46.469,158.760
C04947=1027.190,184.648,387.343,169.043,46.472,158.760
C04948=1027.185,184.400,387.367,169.039,46.476,158.761
C04949=1027.179,184.151,387.390,169.036,46.479,158.761
C04950=1027.173,183.902,387.413,169.032,46.482,158.761
C04951=1027.168,183.653,387.437,169.028,46.485,158.761
C04952=1027.162,183.404,387.461,169.025,46.488,158.761
C04953=1027.157,183.155,387.485,169.022,46.491,158.762
C04954=1027.151,182.906,387.508,169.018,46.495,158.762
C04955=1027.145,182.657,387.531,169.015,46.498,158.762
C04956=1027.139,182.409,387.554,169.011,46.501,158.762
C04957=1027.133,182.160,387.577,169.008,46.505,158.763
C04958=1027.127,181.911,387.601,169.004,46.508,158.763
C04959=1027.121,181.662,387.624,169.000,46.512,158.763
C04960=1027.115,181.413,387.646,168.997,46.515,158.764
C04961=1027.109,181.164,387.669,168.993,46.519,158.764
C04962=1027.103,180.915,387.692,168.990,46.522,158.764
C04963=1027.098,180.666,387.715,168.987,46.525,158.765
C04964=1027.090,180.417,387.738,168.983,46.528,158.765
C04965=1027.085,180.168,387.761,168.980,46.532,158.765
C04966=1027.079,179.919,387.783,168.976,46.535,158.765
C04967=1027.073,179.671,387.807,168.973,46.539,158.766
C04968=1027.067,179.423,387.829,168.970,46.542,158.766
C04969=1027.061,179.174,387.852,168.966,46.546,158.766
C04970=1027.055,178.925,387.875,168.962,46.549,158.766
C04971=1027.049,178.676,387.898,168.959,46.553,158.767
C04972=1027.043,178.426,387.922,168.955,46.556,158.767
C04973=1027.037,178.178,387.944,168.952,46.559,158.767
C04974=1027.031,177.929,387.967,168.948,46.563,158.767
C04975=1027.025,177.680,387.990,168.945,46.566,158.768
C04976=1027.019,177.431,388.013,168.942,46.570,158.768
C04977=1027.013,177.182,388.035,168.938,46.573,158.768
C04978=1027.007,176.933,388.058,168.935,46.577,158.769
C04979=1027.002,176.684,388.080,168.932,46.580,158.769
C04980=1026.996,176.435,388.103,168.928,46.584,158.769
C04981=1026.989,176.186,388.126,168.925,46.587,158.770
C04982=1026.984,175.938,388.149,168.921,46.591,158.770
C04983=1026.978,175.689,388.172,168.918,46.594,158.770
C04984=1026.972,175.440,388.194,168.915,46.597,158.771
C04985=1026.966,175.191,388.217,168.911,46.601,158.771
C04986=1026.960,174.942,388.240,168.908,46.604,158.771
C04987=1026.954,174.693,388.263,168.904,46.607,158.771
C04988=1026.949,174.445,388.286,168.902,46.611,158.772
C04989=1026.942,174.195,388.307,168.897,46.614,158.772
C04990=1026.937,173.946,388.330,168.894,46.618,158.772
C04991=1026.931,173.698,388.353,168.891,46.622,158.773
C04992=1026.925,173.449,388.376,168.887,46.625,158.773
C04993=1026.919,173.200,388.398,168.884,46.628,158.773
C04994=1026.913,172.951,388.421,168.881,46.631,158.773
C04995=1026.908,172.702,388.444,168.877,46.635,158.774
C04996=1026.901,172.419,388.470,168.874,46.639,158.774
C04997=1026.894,172.135,388.496,168.870,46.643,158.774
C04998=1026.887,171.852,388.520,168.866,46.647,158.775
C04999=1026.881,171.569,388.546,168.862,46.651,158.775
C05000=1026.875,171.320,388.569,168.859,46.654,158.775
C05001=1026.870,171.070,388.592,168.855,46.658,158.776
C05002=1026.864,170.822,388.615,168.852,46.661,158.776
C05003=1026.858,170.573,388.637,168.849,46.664,158.776
C05004=1026.852,170.324,388.660,168.846,46.668,158.777
C05005=1026.846,170.075,388.682,168.842,46.671,158.777
C05006=1026.840,169.826,388.704,168.839,46.675,158.777
C05007=1026.835,169.578,388.727,168.836,46.678,158.777
C05008=1026.829,169.328,388.749,168.833,46.682,158.778
C05009=1026.824,169.079,388.772,168.829,46.685,158.778
C05010=1026.817,168.831,388.795,168.826,46.689,158.778
C05011=1026.812,168.581,388.817,168.823,46.692,158.779
C05012=1026.806,168.332,388.840,168.820,46.695,158.779
C05013=1026.800,168.084,388.862,168.817,46.699,158.779
C05014=1026.795,167.835,388.884,168.813,46.702,158.779
C05015=1026.789,167.586,388.907,168.810,46.706,158.780
C05016=1026.784,167.337,388.929,168.807,46.709,158.780
C05017=1026.777,167.088,388.952,168.804,46.713,158.780
C05018=1026.771,166.839,388.974,168.800,46.716,158.781
C05019=1026.766,166.590,388.997,168.797,46.720,158.781
C05020=1026.760,166.342,389.019,168.794,46.723,158.781
C05021=1026.755,166.092,389.041,168.790,46.726,158.782
C05022=1026.749,165.843,389.064,168.787,46.730,158.782
C05023=1026.743,165.594,389.086,168.784,46.733,158.782
C05024=1026.738,165.346,389.108,168.780,46.737,158.782
C05025=1026.732,165.096,389.130,168.777,46.740,158.783
C05026=1026.726,164.847,389.153,168.774,46.744,158.783
C05027=1026.720,164.599,389.176,168.771,46.747,158.783
C05028=1026.715,164.349,389.198,168.768,46.750,158.784
C05029=1026.709,164.101,389.220,168.765,46.754,158.784
C05030=1026.703,163.852,389.242,168.762,46.757,158.784
C05031=1026.698,163.603,389.265,168.758,46.761,158.785
C05032=1026.693,163.354,389.287,168.755,46.764,158.785
C05033=1026.687,163.105,389.309,168.752,46.768,158.785
C05034=1026.681,162.856,389.331,168.749,46.771,158.785
C05035=1026.675,162.607,389.354,168.746,46.774,158.786
C05036=1026.670,162.358,389.376,168.743,46.778,158.786
C05037=1026.664,162.109,389.398,168.740,46.781,158.786
C05038=1026.658,161.860,389.421,168.736,46.785,158.787
C05039=1026.654,161.611,389.443,168.733,46.788,158.787
C05040=1026.647,161.362,389.464,168.730,46.792,158.787
C05041=1026.642,161.113,389.487,168.727,46.795,158.787
C05042=1026.637,160.865,389.509,168.724,46.798,158.788
C05043=1026.630,160.616,389.531,168.721,46.802,158.788
C05044=1026.625,160.366,389.554,168.718,46.805,158.788
C05045=1026.620,160.118,389.576,168.715,46.809,158.789
C05046=1026.614,159.869,389.599,168.711,46.812,158.789
C05047=1026.608,159.620,389.620,168.709,46.816,158.789
C05048=1026.603,159.371,389.642,168.704,46.819,158.790
C05049=1026.597,159.122,389.664,168.701,46.823,158.790
C05050=1026.591,158.873,389.686,168.699,46.826,158.790
C05051=1026.585,158.623,389.708,168.696,46.830,158.791
C05052=1026.580,158.375,389.729,168.692,46.833,158.791
C05053=1026.574,158.126,389.751,168.690,46.837,158.791
C05054=1026.567,157.877,389.773,168.686,46.841,158.792
C05055=1026.563,157.628,389.795,168.683,46.844,158.792
C05056=1026.556,157.378,389.816,168.680,46.848,158.792
C05057=1026.550,157.130,389.839,168.677,46.851,158.793
C05058=1026.544,156.881,389.860,168.674,46.855,158.793
C05059=1026.539,156.632,389.882,168.671,46.858,158.793
C05060=1026.532,156.348,389.906,168.667,46.862,158.794
C05061=1026.526,156.064,389.931,168.663,46.867,158.794
C05062=1026.519,155.781,389.956,168.660,46.871,158.795
C05063=1026.512,155.497,389.980,168.656,46.875,158.795
C05064=1026.507,155.247,390.002,168.654,46.878,158.795
C05065=1026.501,154.999,390.024,168.651,46.882,158.796
C05066=1026.495,154.749,390.045,168.647,46.886,158.796
C05067=1026.490,154.501,390.067,168.644,46.889,158.796
C05068=1026.484,154.251,390.089,168.641,46.893,158.797
C05069=1026.478,154.002,390.110,168.638,46.897,158.797
C05070=1026.472,153.754,390.132,168.635,46.900,158.797
C05071=1026.466,153.504,390.153,168.632,46.904,158.798
C05072=1026.461,153.256,390.175,168.629,46.907,158.798
C05073=1026.454,153.007,390.196,168.626,46.911,158.798
C05074=1026.449,152.757,390.218,168.623,46.914,158.799
C05075=1026.444,152.509,390.240,168.619,46.918,158.799
C05076=1026.437,152.260,390.261,168.616,46.922,158.799
C05077=1026.432,152.011,390.283,168.613,46.926,158.800
C05078=1026.426,151.762,390.304,168.610,46.929,158.800
C05079=1026.420,151.512,390.325,168.607,46.932,158.800
C05080=1026.414,151.263,390.346,168.604,46.936,158.801
C05081=1026.408,151.014,390.368,168.601,46.940,158.801
C05082=1026.402,150.766,390.389,168.598,46.944,158.801
C05083=1026.396,150.517,390.411,168.596,46.947,158.802
C05084=1026.391,150.268,390.432,168.592,46.951,158.802
C05085=1026.385,150.018,390.453,168.589,46.955,158.803
C05086=1026.379,149.770,390.474,168.586,46.958,158.803
C05087=1026.374,149.520,390.497,168.583,46.962,158.803
C05088=1026.368,149.272,390.518,168.580,46.965,158.804
C05089=1026.362,149.022,390.540,168.577,46.969,158.804
C05090=1026.357,148.773,390.560,168.574,46.973,158.804
C05091=1026.351,148.524,390.582,168.571,46.977,158.805
C05092=1026.345,148.276,390.603,168.568,46.980,158.805
C05093=1026.339,148.026,390.625,168.565,46.984,158.805
C05094=1026.334,147.777,390.645,168.562,46.987,158.806
C05095=1026.328,147.528,390.667,168.559,46.991,158.806
C05096=1026.322,147.280,390.688,168.556,46.995,158.806
C05097=1026.316,147.030,390.709,168.552,46.998,158.807
C05098=1026.311,146.781,390.730,168.550,47.002,158.807
C05099=1026.304,146.532,390.752,168.547,47.006,158.807
C05100=1026.299,146.283,390.773,168.544,47.010,158.808
C05101=1026.293,146.034,390.794,168.541,47.013,158.808
C05102=1026.287,145.786,390.815,168.538,47.017,158.809
C05103=1026.281,145.536,390.836,168.535,47.021,158.809
C05104=1026.275,145.287,390.857,168.532,47.025,158.809
C05105=1026.269,145.037,390.878,168.529,47.028,158.810
C05106=1026.264,144.789,390.899,168.526,47.032,158.810
C05107=1026.257,144.540,390.920,168.523,47.035,158.810
C05108=1026.252,144.291,390.941,168.520,47.039,158.811
C05109=1026.246,144.042,390.962,168.517,47.042,158.811
C05110=1026.240,143.793,390.983,168.514,47.046,158.811
C05111=1026.234,143.543,391.005,168.511,47.050,158.812
C05112=1026.228,143.295,391.025,168.508,47.054,158.812
C05113=1026.223,143.046,391.046,168.505,47.058,158.812
C05114=1026.217,142.796,391.067,168.502,47.061,158.813
C05115=1026.211,142.548,391.088,168.499,47.065,158.813
C05116=1026.205,142.298,391.109,168.496,47.069,158.814
C05117=1026.199,142.050,391.130,168.493,47.073,158.814
C05118=1026.193,141.800,391.151,168.490,47.076,158.814
C05119=1026.188,141.551,391.172,168.488,47.080,158.815
C05120=1026.182,141.302,391.192,168.485,47.084,158.815
C05121=1026.177,141.052,391.213,168.482,47.087,158.815
C05122=1026.170,140.804,391.234,168.479,47.091,158.816
C05123=1026.165,140.555,391.255,168.476,47.095,158.816
C05124=1026.158,140.271,391.279,168.472,47.099,158.817
C05125=1026.152,139.987,391.303,168.469,47.103,158.817
C05126=1026.145,139.703,391.327,168.466,47.107,158.817
C05127=1026.138,139.418,391.350,168.463,47.112,158.818
C05128=1026.133,139.170,391.371,168.460,47.115,158.818
C05129=1026.127,138.920,391.392,168.457,47.119,158.819
C05130=1026.121,138.671,391.413,168.454,47.123,158.819
C05131=1026.115,138.423,391.433,168.451,47.127,158.819
C05132=1026.110,138.173,391.454,168.449,47.130,158.820
C05133=1026.104,137.924,391.475,168.446,47.134,158.820
C05134=1026.098,137.675,391.495,168.442,47.138,158.820
C05135=1026.092,137.426,391.516,168.439,47.142,158.821
C05136=1026.086,137.177,391.536,168.436,47.146,158.821
C05137=1026.081,136.928,391.558,168.433,47.149,158.822
C05138=1026.075,136.679,391.578,168.430,47.153,158.822
C05139=1026.069,136.430,391.598,168.427,47.157,158.822
C05140=1026.064,136.181,391.619,168.425,47.160,158.823
C05141=1026.057,135.931,391.639,168.422,47.164,158.823
C05142=1026.051,135.683,391.661,168.419,47.168,158.823
C05143=1026.045,135.434,391.681,168.416,47.172,158.824
C05144=1026.039,135.184,391.701,168.413,47.175,158.824
C05145=1026.034,134.935,391.722,168.410,47.179,158.825
C05146=1026.028,134.686,391.742,168.407,47.183,158.825
C05147=1026.022,134.437,391.764,168.404,47.187,158.825
C05148=1026.016,134.188,391.784,168.401,47.190,158.826
C05149=1026.011,133.939,391.804,168.399,47.194,158.826
C05150=1026.005,133.690,391.824,168.396,47.198,158.826
C05151=1025.999,133.440,391.845,168.393,47.202,158.827
C05152=1025.993,133.191,391.865,168.390,47.206,158.827
C05153=1025.988,132.942,391.885,168.387,47.210,158.828
C05154=1025.981,132.693,391.906,168.384,47.214,158.828
C05155=1025.976,132.444,391.926,168.382,47.217,158.828
C05156=1025.970,132.195,391.947,168.379,47.221,158.829
C05157=1025.964,131.946,391.968,168.376,47.225,158.829
C05158=1025.958,131.697,391.988,168.373,47.229,158.830
C05159=1025.952,131.448,392.008,168.370,47.232,158.830
C05160=1025.946,131.199,392.028,168.367,47.236,158.830
C05161=1025.941,130.950,392.049,168.365,47.239,158.831
C05162=1025.935,130.701,392.069,168.362,47.243,158.831
C05163=1025.929,130.451,392.090,168.360,47.247,158.832
C05164=1025.923,130.202,392.110,168.357,47.251,158.832
C05165=1025.918,129.953,392.130,168.354,47.254,158.832
C05166=1025.912,129.704,392.150,168.351,47.258,158.833
C05167=1025.906,129.455,392.171,168.348,47.263,158.833
C05168=1025.900,129.206,392.191,168.345,47.267,158.833
C05169=1025.894,128.957,392.210,168.342,47.270,158.834
C05170=1025.889,128.707,392.230,168.339,47.274,158.834
C05171=1025.882,128.458,392.251,168.336,47.278,158.835
C05172=1025.876,128.209,392.271,168.333,47.282,158.835
C05173=1025.870,127.960,392.291,168.330,47.286,158.836
C05174=1025.864,127.712,392.311,168.328,47.290,158.836
C05175=1025.857,127.462,392.331,168.325,47.294,158.836
C05176=1025.852,127.212,392.351,168.322,47.297,158.837
C05177=1025.846,126.963,392.371,168.319,47.302,158.837
C05178=1025.840,126.715,392.391,168.316,47.306,158.838
C05179=1025.834,126.466,392.411,168.314,47.309,158.838
C05180=1025.828,126.216,392.431,168.311,47.313,158.838
C05181=1025.823,125.967,392.451,168.308,47.317,158.839
C05182=1025.817,125.718,392.471,168.305,47.321,158.839
C05183=1025.811,125.469,392.491,168.302,47.325,158.840
C05184=1025.805,125.220,392.511,168.299,47.329,158.840
C05185=1025.799,124.971,392.530,168.297,47.333,158.840
C05186=1025.793,124.721,392.550,168.294,47.336,158.841
C05187=1025.787,124.472,392.571,168.291,47.340,158.841
C05188=1025.778,124.062,392.604,168.287,47.346,158.842
C05189=1025.768,123.652,392.636,168.282,47.353,158.842
C05190=1025.758,123.242,392.669,168.278,47.359,158.843
C05191=1025.749,122.831,392.702,168.273,47.366,158.844
C05192=1025.743,122.583,392.722,168.270,47.370,158.844
C05193=1025.737,122.334,392.741,168.267,47.373,158.844
C05194=1025.732,122.084,392.761,168.265,47.377,158.845
C05195=1025.726,121.835,392.781,168.262,47.381,158.845
C05196=1025.720,121.586,392.801,168.260,47.384,158.846
C05197=1025.714,121.337,392.820,168.257,47.389,158.846
C05198=1025.708,121.088,392.840,168.254,47.393,158.847
C05199=1025.702,120.838,392.860,168.251,47.396,158.847
C05200=1025.696,120.589,392.881,168.248,47.400,158.847
C05201=1025.690,120.340,392.901,168.245,47.404,158.848
C05202=1025.685,120.091,392.920,168.243,47.408,158.848
C05203=1025.679,119.842,392.940,168.240,47.411,158.848
C05204=1025.673,119.593,392.960,168.237,47.415,158.849
C05205=1025.667,119.344,392.979,168.234,47.420,158.849
C05206=1025.661,119.095,392.999,168.231,47.423,158.850
C05207=1025.656,118.845,393.019,168.229,47.427,158.850
C05208=1025.650,118.596,393.039,168.227,47.431,158.851
C05209=1025.644,118.347,393.059,168.224,47.434,158.851
C05210=1025.638,118.098,393.078,168.221,47.438,158.851
C05211=1025.632,117.849,393.098,168.218,47.442,158.852
C05212=1025.627,117.600,393.117,168.215,47.446,158.852
C05213=1025.621,117.351,393.138,168.212,47.450,158.852
C05214=1025.616,117.101,393.157,168.210,47.453,158.853
C05215=1025.610,116.852,393.177,168.207,47.458,158.853
C05216=1025.604,116.603,393.196,168.204,47.462,158.854
C05217=1025.598,116.354,393.216,168.202,47.465,158.854
C05218=1025.592,116.105,393.235,168.199,47.469,158.854
C05219=1025.586,115.856,393.255,168.197,47.473,158.855
C05220=1025.581,115.606,393.275,168.194,47.476,158.855
C05221=1025.575,115.357,393.295,168.191,47.480,158.856
C05222=1025.570,115.108,393.314,168.188,47.484,158.856
C05223=1025.564,114.859,393.334,168.185,47.488,158.856
C05224=1025.558,114.610,393.354,168.182,47.492,158.857
C05225=1025.552,114.361,393.373,168.180,47.495,158.857
C05226=1025.546,114.111,393.393,168.178,47.499,158.857
C05227=1025.540,113.863,393.413,168.175,47.503,158.858
C05228=1025.535,113.613,393.433,168.172,47.507,158.858
C05229=1025.529,113.364,393.452,168.169,47.511,158.859
C05230=1025.524,113.115,393.472,168.167,47.515,158.859
C05231=1025.518,112.865,393.491,168.164,47.518,158.859
C05232=1025.512,112.616,393.511,168.162,47.522,158.860
C05233=1025.506,112.367,393.530,168.159,47.526,158.860
C05234=1025.501,112.117,393.549,168.156,47.529,158.861
C05235=1025.495,111.869,393.569,168.153,47.533,158.861
C05236=1025.486,111.496,393.598,168.149,47.540,158.862
C05237=1025.477,111.124,393.626,168.145,47.545,158.862
C05238=1025.469,110.752,393.656,168.141,47.551,158.863
C05239=1025.460,110.379,393.684,168.137,47.556,158.863
C05240=1025.454,110.130,393.704,168.135,47.561,158.864
C05241=1025.448,109.881,393.723,168.132,47.565,158.864
C05242=1025.442,109.632,393.742,168.129,47.568,158.865
C05243=1025.436,109.382,393.761,168.126,47.572,158.865
C05244=1025.431,109.133,393.780,168.124,47.577,158.866
C05245=1025.424,108.884,393.799,168.121,47.580,158.866
C05246=1025.418,108.635,393.819,168.118,47.584,158.866
C05247=1025.413,108.385,393.838,168.115,47.588,158.867
C05248=1025.406,108.101,393.859,168.113,47.592,158.867
C05249=1025.399,107.816,393.881,168.109,47.597,158.868
C05250=1025.392,107.532,393.903,168.107,47.602,158.868
C05251=1025.386,107.249,393.925,168.103,47.606,158.869
C05252=1025.380,106.999,393.944,168.100,47.610,158.869
C05253=1025.374,106.750,393.963,168.098,47.614,158.869
C05254=1025.368,106.501,393.982,168.096,47.618,158.870
C05255=1025.362,106.251,394.001,168.093,47.622,158.870
C05256=1025.356,106.002,394.020,168.090,47.626,158.871
C05257=1025.350,105.753,394.039,168.087,47.630,158.871
C05258=1025.344,105.503,394.058,168.085,47.634,158.872
C05259=1025.339,105.255,394.077,168.082,47.638,158.872
C05260=1025.333,105.005,394.096,168.079,47.642,158.872
C05261=1025.327,104.756,394.115,168.076,47.645,158.873
C05262=1025.321,104.507,394.134,168.074,47.649,158.873
C05263=1025.315,104.257,394.153,168.072,47.653,158.874
C05264=1025.309,104.008,394.172,168.069,47.657,158.874
C05265=1025.303,103.759,394.191,168.066,47.661,158.874
C05266=1025.298,103.510,394.210,168.063,47.665,158.875
C05267=1025.292,103.261,394.229,168.060,47.669,158.875
C05268=1025.286,103.011,394.248,168.058,47.673,158.876
C05269=1025.280,102.762,394.267,168.055,47.677,158.876
C05270=1025.274,102.513,394.286,168.053,47.680,158.876
C05271=1025.269,102.264,394.305,168.050,47.684,158.877
C05272=1025.263,102.015,394.324,168.048,47.688,158.877
C05273=1025.257,101.766,394.343,168.045,47.693,158.878
C05274=1025.251,101.516,394.362,168.042,47.696,158.878
C05275=1025.245,101.267,394.381,168.039,47.700,158.878
C05276=1025.240,101.018,394.399,168.036,47.704,158.879
C05277=1025.234,100.769,394.419,168.035,47.708,158.879
C05278=1025.228,100.519,394.438,168.032,47.712,158.880
C05279=1025.222,100.270,394.457,168.029,47.716,158.880
C05280=1025.216,100.021,394.476,168.026,47.720,158.880
C05281=1025.211,99.772,394.495,168.024,47.723,158.881
C05282=1025.205,99.522,394.513,168.021,47.727,158.881
C05283=1025.198,99.273,394.531,168.019,47.731,158.882
C05284=1025.193,99.024,394.551,168.016,47.735,158.882
C05285=1025.186,98.775,394.569,168.014,47.739,158.882
C05286=1025.181,98.526,394.588,168.011,47.743,158.883
C05287=1025.175,98.276,394.606,168.008,47.747,158.883
C05288=1025.169,98.027,394.625,168.005,47.751,158.884
C05289=1025.163,97.778,394.644,168.002,47.755,158.884
C05290=1025.157,97.529,394.663,168.000,47.759,158.885
C05291=1025.151,97.280,394.680,167.997,47.763,158.885
C05292=1025.145,97.030,394.699,167.994,47.767,158.885
C05293=1025.139,96.781,394.718,167.993,47.771,158.886
C05294=1025.133,96.532,394.737,167.990,47.775,158.886
C05295=1025.128,96.283,394.755,167.987,47.779,158.887
C05296=1025.121,96.033,394.773,167.984,47.783,158.887
C05297=1025.116,95.784,394.793,167.982,47.787,158.888
C05298=1025.110,95.535,394.810,167.979,47.791,158.888
C05299=1025.104,95.286,394.829,167.976,47.795,158.888
C05300=1025.098,95.036,394.848,167.973,47.799,158.889
C05301=1025.092,94.787,394.866,167.972,47.803,158.889
C05302=1025.086,94.538,394.884,167.969,47.807,158.890
C05303=1025.080,94.289,394.904,167.966,47.811,158.890
C05304=1025.074,94.039,394.922,167.963,47.815,158.890
C05305=1025.069,93.790,394.941,167.961,47.819,158.891
C05306=1025.063,93.541,394.959,167.958,47.823,158.891
C05307=1025.057,93.291,394.977,167.955,47.826,158.892
C05308=1025.051,93.042,394.996,167.953,47.830,158.892
C05309=1025.045,92.793,395.014,167.951,47.835,158.893
C05310=1025.039,92.544,395.032,167.948,47.838,158.893
C05311=1025.033,92.294,395.052,167.945,47.842,158.893
C05312=1025.027,92.010,395.072,167.942,47.847,158.894
C05313=1025.020,91.726,395.093,167.939,47.851,158.894
C05314=1025.013,91.442,395.115,167.936,47.856,158.895
C05315=1025.006,91.158,395.136,167.934,47.860,158.895
C05316=1025.001,90.909,395.153,167.931,47.864,158.896
C05317=1024.995,90.659,395.172,167.928,47.868,158.896
C05318=1024.989,90.409,395.190,167.925,47.872,158.896
C05319=1024.983,90.161,395.209,167.923,47.876,158.897
C05320=1024.978,89.911,395.227,167.920,47.880,158.897
C05321=1024.971,89.662,395.246,167.918,47.884,158.898
C05322=1024.966,89.413,395.263,167.915,47.888,158.898
C05323=1024.960,89.163,395.283,167.913,47.891,158.898
C05324=1024.954,88.914,395.301,167.910,47.895,158.899
C05325=1024.948,88.665,395.319,167.907,47.900,158.899
C05326=1024.942,88.415,395.337,167.904,47.904,158.900
C05327=1024.936,88.166,395.355,167.902,47.908,158.900
C05328=1024.930,87.917,395.373,167.899,47.912,158.901
C05329=1024.924,87.668,395.391,167.897,47.915,158.901
C05330=1024.919,87.418,395.409,167.895,47.920,158.901
C05331=1024.912,87.169,395.427,167.892,47.924,158.902
C05332=1024.906,86.920,395.445,167.889,47.928,158.902
C05333=1024.900,86.671,395.463,167.887,47.932,158.903
C05334=1024.894,86.421,395.481,167.884,47.936,158.903
C05335=1024.888,86.172,395.499,167.881,47.940,158.903
C05336=1024.882,85.923,395.517,167.878,47.944,158.904
C05337=1024.876,85.674,395.535,167.876,47.948,158.904
C05338=1024.870,85.425,395.553,167.874,47.952,158.905
C05339=1024.864,85.175,395.571,167.871,47.956,158.905
C05340=1024.858,84.926,395.590,167.868,47.960,158.906
C05341=1024.852,84.677,395.607,167.866,47.964,158.906
C05342=1024.846,84.427,395.625,167.863,47.968,158.906
C05343=1024.840,84.178,395.643,167.860,47.972,158.907
C05344=1024.834,83.929,395.661,167.857,47.976,158.907
C05345=1024.830,83.679,395.679,167.856,47.980,158.908
C05346=1024.823,83.430,395.697,167.853,47.984,158.908
C05347=1024.817,83.181,395.716,167.850,47.988,158.909
C05348=1024.811,82.931,395.734,167.847,47.992,158.909
C05349=1024.805,82.682,395.752,167.845,47.996,158.909
C05350=1024.800,82.433,395.769,167.842,48.000,158.910
C05351=1024.793,82.184,395.788,167.840,48.004,158.910
C05352=1024.788,81.935,395.805,167.838,48.008,158.911
C05353=1024.782,81.685,395.823,167.835,48.011,158.911
C05354=1024.776,81.436,395.841,167.832,48.016,158.911
C05355=1024.770,81.186,395.859,167.829,48.020,158.912
C05356=1024.764,80.938,395.877,167.827,48.024,158.912
C05357=1024.758,80.688,395.895,167.825,48.027,158.913
C05358=1024.753,80.439,395.913,167.822,48.032,158.913
C05359=1024.747,80.189,395.931,167.819,48.036,158.913
C05360=1024.741,79.940,395.948,167.817,48.039,158.914
C05361=1024.735,79.691,395.967,167.814,48.043,158.914
C05362=1024.729,79.442,395.984,167.811,48.048,158.915
C05363=1024.723,79.192,396.002,167.809,48.051,158.915
C05364=1024.717,78.943,396.020,167.807,48.055,158.915
C05365=1024.711,78.693,396.038,167.804,48.059,158.916
C05366=1024.706,78.444,396.055,167.801,48.063,158.916
C05367=1024.700,78.195,396.073,167.799,48.067,158.917
C05368=1024.694,77.946,396.091,167.797,48.071,158.917
C05369=1024.688,77.696,396.109,167.794,48.075,158.917
C05370=1024.682,77.447,396.127,167.791,48.079,158.918
C05371=1024.676,77.198,396.145,167.789,48.083,158.918
C05372=1024.671,76.949,396.162,167.786,48.087,158.919
C05373=1024.664,76.699,396.180,167.783,48.091,158.919
C05374=1024.658,76.450,396.197,167.780,48.095,158.919
C05375=1024.652,76.200,396.215,167.779,48.099,158.920
C05376=1024.646,75.916,396.235,167.775,48.104,158.920
C05377=1024.639,75.632,396.256,167.773,48.108,158.921
C05378=1024.632,75.348,396.275,167.769,48.113,158.921
C05379=1024.625,75.063,396.296,167.766,48.117,158.922
C05380=1024.620,74.814,396.313,167.764,48.122,158.922
C05381=1024.613,74.565,396.330,167.761,48.125,158.923
C05382=1024.607,74.316,396.348,167.758,48.129,158.923
C05383=1024.602,74.066,396.366,167.757,48.134,158.924
C05384=1024.596,73.817,396.384,167.754,48.137,158.924
C05385=1024.590,73.567,396.400,167.751,48.141,158.924
C05386=1024.584,73.318,396.418,167.749,48.146,158.925
C05387=1024.578,73.069,396.435,167.746,48.150,158.925
C05388=1024.572,72.819,396.453,167.743,48.154,158.926
C05389=1024.566,72.570,396.470,167.740,48.157,158.926
C05390=1024.560,72.321,396.488,167.739,48.162,158.926
C05391=1024.554,72.071,396.506,167.736,48.166,158.927
C05392=1024.548,71.823,396.523,167.733,48.169,158.927
C05393=1024.542,71.572,396.540,167.730,48.173,158.928
C05394=1024.537,71.323,396.557,167.728,48.178,158.928
C05395=1024.531,71.074,396.575,167.725,48.182,158.928
C05396=1024.524,70.825,396.592,167.723,48.185,158.929
C05397=1024.519,70.576,396.610,167.721,48.190,158.929
C05398=1024.513,70.327,396.628,167.718,48.194,158.930
C05399=1024.507,70.077,396.644,167.715,48.197,158.930
C05400=1024.501,69.828,396.662,167.712,48.201,158.930
C05401=1024.495,69.578,396.680,167.710,48.206,158.931
C05402=1024.489,69.329,396.697,167.708,48.209,158.931
C05403=1024.483,69.080,396.714,167.705,48.213,158.932
C05404=1024.477,68.830,396.731,167.702,48.217,158.932
C05405=1024.472,68.581,396.749,167.700,48.222,158.933
C05406=1024.466,68.332,396.766,167.697,48.226,158.933
C05407=1024.460,68.082,396.783,167.694,48.229,158.933
C05408=1024.454,67.833,396.800,167.692,48.234,158.934
C05409=1024.448,67.584,396.818,167.690,48.238,158.934
C05410=1024.441,67.334,396.835,167.687,48.241,158.935
C05411=1024.436,67.085,396.852,167.684,48.245,158.935
C05412=1024.430,66.836,396.869,167.682,48.250,158.935
C05413=1024.424,66.586,396.887,167.679,48.254,158.936
C05414=1024.418,66.337,396.903,167.676,48.258,158.936
C05415=1024.412,66.088,396.921,167.674,48.262,158.937
C05416=1024.406,65.837,396.938,167.672,48.266,158.937
C05417=1024.400,65.589,396.955,167.669,48.270,158.937
C05418=1024.394,65.340,396.972,167.667,48.274,158.938
C05419=1024.388,65.090,396.989,167.664,48.278,158.938
C05420=1024.382,64.841,397.007,167.661,48.282,158.939
C05421=1024.376,64.592,397.024,167.658,48.286,158.939
C05422=1024.370,64.342,397.041,167.656,48.290,158.940
C05423=1024.364,64.093,397.058,167.654,48.294,158.940
C05424=1024.359,63.843,397.075,167.651,48.298,158.940
C05425=1024.352,63.594,397.092,167.649,48.302,158.941
C05426=1024.347,63.344,397.109,167.646,48.306,158.941
C05427=1024.341,63.095,397.126,167.643,48.310,158.942
C05428=1024.334,62.845,397.142,167.641,48.315,158.942
C05429=1024.328,62.597,397.159,167.638,48.319,158.942
C05430=1024.323,62.347,397.176,167.635,48.323,158.943
C05431=1024.317,62.098,397.192,167.633,48.327,158.943
C05432=1024.310,61.848,397.210,167.631,48.331,158.944
C05433=1024.304,61.599,397.226,167.628,48.335,158.944
C05434=1024.298,61.350,397.243,167.626,48.339,158.945
C05435=1024.292,61.100,397.260,167.623,48.344,158.945
C05436=1024.285,60.851,397.277,167.620,48.347,158.945
C05437=1024.279,60.602,397.293,167.618,48.352,158.946
C05438=1024.274,60.352,397.310,167.615,48.356,158.946
C05439=1024.267,60.103,397.327,167.612,48.360,158.947
C05440=1024.260,59.819,397.346,167.610,48.364,158.947
C05441=1024.253,59.534,397.365,167.606,48.369,158.948
C05442=1024.246,59.249,397.384,167.604,48.374,158.948
C05443=1024.240,58.965,397.404,167.600,48.379,158.948
C05444=1024.234,58.716,397.420,167.598,48.383,158.949
C05445=1024.227,58.466,397.436,167.595,48.387,158.949
C05446=1024.221,58.217,397.453,167.594,48.391,158.950
C05447=1024.215,57.967,397.470,167.591,48.395,158.950
C05448=1024.209,57.718,397.486,167.588,48.399,158.951
C05449=1024.204,57.469,397.503,167.585,48.404,158.951
C05450=1024.197,57.219,397.520,167.583,48.408,158.952
C05451=1024.191,56.970,397.536,167.580,48.412,158.952
C05452=1024.185,56.721,397.553,167.577,48.416,158.952
C05453=1024.179,56.472,397.570,167.575,48.420,158.953
C05454=1024.174,56.222,397.586,167.572,48.424,158.953
C05455=1024.167,55.972,397.603,167.569,48.428,158.954
C05456=1024.161,55.723,397.620,167.568,48.432,158.954
C05457=1024.155,55.474,397.636,167.565,48.436,158.954
C05458=1024.149,55.224,397.653,167.562,48.441,158.955
